# B&R Automation Studio project 2x1HWDemo
Automation Studio 4.9.2.46; technology packages: mapp 5.14.0, mappCockpit 5.14.0, mappControl 5.14.0, mappMotion 5.14.0, mappView 5.14.0

## Configuration 1685

CPU X20CP1685, AutomationRuntime C4.90, Build 6.3.0, Safety 1.10, Vc V4.72.2

### Task classes (Cpu.sw)
```
Cyclic#1 (cycle 1000 us, tolerance 0 us):
  6DCtrl <- Source.6DCtrl.6DCtrl.prg
  RbtCtrl <- Source.Robot.RbtCtrl.prg
  ShCtrl <- Source.ShuttleCtrl.ShCtrl.prg
Cyclic#2 (cycle 10000 us, tolerance 10000 us):
  Main <- Source.Main.Main.prg
Cyclic#4:
  Recovery <- Source.ShuttleCtrl.Recovery.prg
Cyclic#8 (cycle 1000 us):
  Vis <- Source.Auxil.Vis.prg
  AuditCtrl <- Source.Auxil.AuditCtrl.prg
  MacroLoad <- Source.6DCtrl.MacroLoad.prg
DataObjects: McAcpSys
Binaries: mvLoader, arcoal, McMechSys, arflatprv, arsvcreg, McProfGen, TCData, McAcpSim, mCoWebSc, FWRules, McAcpDrv, udbdef, Role, Config_3, arconfig, Settings, User, asfw, ashwd, Config_1, ashwac, sysconf, Config_4, Config, Hierarchy, Config_2, iomap
Libraries: McBase, McAxis, MpBase, AsMath, AsXml, operator, runtime, astime, AsIecCon, standard, AsBrStr, AsIODiag, LoggingLib, asstring, ArEventLog, AsTCP, FileIO, snprintf, brsystem, AsZip, MTTypes, sys_lib, CoTrace, McAcpAx, McPathGen, McAcpTrak, McAxGroup, McProgInt, MpRobotics, MTBasics, McAcp6D, MpAudit, asarlog, asepl, asmem, aruser, dataobj, powerlnk, asarprof, arssl
```

### Hardware
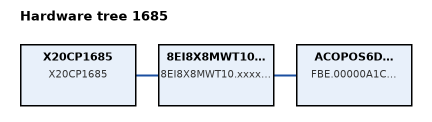
```
8EI8X8MWT10.xxxx-1 : 8EI8X8MWT10.xxxx-1 v2.3.0.2  [PLK1 -> X20CP1685.IF3 (NodeNumber=2) [Cable Type=PowerlinkCable, Length=10, Version=1.0.0.3]; PLK2 -> ACOPOS6D_POWERLINK.PLK1 (NodeNumber=2) [Cable Type=PowerlinkCable, Length=10, Version=1.0.0.3]]
  DriveConfiguration/Module:
    McAcoposTypeID = AcoposP3TConfig
    ActivateACOPOSSimulationOnPLC = 1
  DriveConfiguration/Channel[1]/RealAxis:
    AxisReference = gAxisQ1
  DriveConfiguration/Channel[1]/RealAxis/MechanicalElements/Gearbox:
    InputIsReadOnly = 0
    Input = 1
    OutputIsReadOnly = 0
    Output = 1
  DriveConfiguration/Channel[1]/RealAxis/MechanicalElements/RotaryToLinearTransformation:
    ReferenceDistanceIsReadOnly = 0
    ReferenceDistance = 1
  DriveConfiguration/Channel[1]/RealAxis/Controller:
    ModeIsReadOnly = 0
    Mode = PositionController
  DriveConfiguration/Channel[1]/RealAxis/Controller/Mode/Position:
    ProportionalGain = 50.0
    IntegrationTime = 0.0
    PredictionTime = 0.0004
    TotalDelayTime = 0.0004
  DriveConfiguration/Channel[1]/RealAxis/Controller/Mode/Speed:
    ProportionalGainIsReadOnly = 0
    ProportionalGain = 2.0
    IntegrationTimeIsReadOnly = 0
    IntegrationTime = 0.0
    FilterTimeIsReadOnly = 0
    FilterTime = 0.0
  DriveConfiguration/Channel[1]/RealAxis/Controller/Mode/LoopFilters:
    LoopFilter1 = NotUsed
    LoopFilter2 = NotUsed
    LoopFilter3 = NotUsed
  DriveConfiguration/Channel[1]/RealAxis/Homing:
    Mode = Direct
  DriveConfiguration/Channel[1]/RealAxis/Homing/Mode:
    Position = 0.0
    ReferencePulse = NotUsed
  DriveConfiguration/Channel[1]/RealAxis/Homing:
    RestorePositionVariable = 
  DriveConfiguration/Channel[1]/RealAxis/StopReaction:
    Quickstop = DecelerationLimit
    DriveError = DecelerationLimit
  DriveConfiguration/Channel[1]/RealAxis/MovementErrorLimits:
    PositionError = 1.0
    VelocityErrorMonitoring = Automatic1
  DriveConfiguration/Channel[1]/RealAxis:
    JerkFilter = NotUsed
  DriveConfiguration/Channel[1]/RealAxis/DigitalInputs/HomingSwitch:
    Source = NotUsed
    Level = High
  DriveConfiguration/Channel[1]/RealAxis/DigitalInputs/PositiveLimitSwitch:
    Source = NotUsed
    Level = High
  DriveConfiguration/Channel[1]/RealAxis/DigitalInputs/NegativeLimitSwitch:
    Source = NotUsed
    Level = High
  DriveConfiguration/Channel[1]/RealAxis/DigitalInputs/Trigger1:
    Source = X8Trigger1
    Level = High
  DriveConfiguration/Channel[1]/RealAxis/DigitalInputs/Trigger2:
    Source = X8Trigger2
    Level = High
  DriveConfiguration/Channel[1]/RealAxis/DigitalInputs/Quickstop:
    Input = Trigger2
  DriveConfiguration/Channel[1]/RealAxis/Simulation:
    SimulationModeOnPLC = SetValueGeneration
    SimulationModeOnACOPOS = NotUsed
  DriveConfiguration/Channel[2]/RealAxis:
    AxisReference = gAxisQ2
  DriveConfiguration/Channel[2]/RealAxis/MechanicalElements/Gearbox:
    InputIsReadOnly = 0
    Input = 1
    OutputIsReadOnly = 0
    Output = 1
  DriveConfiguration/Channel[2]/RealAxis/MechanicalElements/RotaryToLinearTransformation:
    ReferenceDistanceIsReadOnly = 0
    ReferenceDistance = 1
  DriveConfiguration/Channel[2]/RealAxis/Controller:
    ModeIsReadOnly = 0
    Mode = PositionController
  DriveConfiguration/Channel[2]/RealAxis/Controller/Mode/Position:
    ProportionalGain = 50.0
    IntegrationTime = 0.0
    PredictionTime = 0.0004
    TotalDelayTime = 0.0004
  DriveConfiguration/Channel[2]/RealAxis/Controller/Mode/Speed:
    ProportionalGainIsReadOnly = 0
    ProportionalGain = 2.0
    IntegrationTimeIsReadOnly = 0
    IntegrationTime = 0.0
    FilterTimeIsReadOnly = 0
    FilterTime = 0.0
  DriveConfiguration/Channel[2]/RealAxis/Controller/Mode/LoopFilters:
    LoopFilter1 = NotUsed
    LoopFilter2 = NotUsed
    LoopFilter3 = NotUsed
  DriveConfiguration/Channel[2]/RealAxis/Homing:
    Mode = Direct
  DriveConfiguration/Channel[2]/RealAxis/Homing/Mode:
    Position = 0.0
    ReferencePulse = NotUsed
  DriveConfiguration/Channel[2]/RealAxis/Homing:
    RestorePositionVariable = 
  DriveConfiguration/Channel[2]/RealAxis/StopReaction:
    Quickstop = DecelerationLimit
    DriveError = DecelerationLimit
  DriveConfiguration/Channel[2]/RealAxis/MovementErrorLimits:
    PositionError = 1.0
    VelocityErrorMonitoring = Automatic1
  DriveConfiguration/Channel[2]/RealAxis:
    JerkFilter = NotUsed
  DriveConfiguration/Channel[2]/RealAxis/DigitalInputs/HomingSwitch:
    Source = NotUsed
    Level = High
  DriveConfiguration/Channel[2]/RealAxis/DigitalInputs/PositiveLimitSwitch:
    Source = NotUsed
    Level = High
  DriveConfiguration/Channel[2]/RealAxis/DigitalInputs/NegativeLimitSwitch:
    Source = NotUsed
    Level = High
  DriveConfiguration/Channel[2]/RealAxis/DigitalInputs/Trigger1:
    Source = X8Trigger1
    Level = High
  DriveConfiguration/Channel[2]/RealAxis/DigitalInputs/Trigger2:
    Source = X8Trigger2
    Level = High
  DriveConfiguration/Channel[2]/RealAxis/DigitalInputs/Quickstop:
    Input = Trigger2
  DriveConfiguration/Channel[2]/RealAxis/Simulation:
    SimulationModeOnPLC = SetValueGeneration
    SimulationModeOnACOPOS = NotUsed
  DriveConfiguration/Channel[3]/RealAxis:
    AxisReference = gAxisQ3
  DriveConfiguration/Channel[3]/RealAxis/MechanicalElements/Gearbox:
    InputIsReadOnly = 0
    Input = 1
    OutputIsReadOnly = 0
    Output = 1
  DriveConfiguration/Channel[3]/RealAxis/MechanicalElements/RotaryToLinearTransformation:
    ReferenceDistanceIsReadOnly = 0
    ReferenceDistance = 1
  DriveConfiguration/Channel[3]/RealAxis/Controller:
    ModeIsReadOnly = 0
    Mode = PositionController
  DriveConfiguration/Channel[3]/RealAxis/Controller/Mode/Position:
    ProportionalGain = 50.0
    IntegrationTime = 0.0
    PredictionTime = 0.0004
    TotalDelayTime = 0.0004
  DriveConfiguration/Channel[3]/RealAxis/Controller/Mode/Speed:
    ProportionalGainIsReadOnly = 0
    ProportionalGain = 2.0
    IntegrationTimeIsReadOnly = 0
    IntegrationTime = 0.0
    FilterTimeIsReadOnly = 0
    FilterTime = 0.0
  DriveConfiguration/Channel[3]/RealAxis/Controller/Mode/LoopFilters:
    LoopFilter1 = NotUsed
    LoopFilter2 = NotUsed
    LoopFilter3 = NotUsed
  DriveConfiguration/Channel[3]/RealAxis/Homing:
    Mode = Direct
  DriveConfiguration/Channel[3]/RealAxis/Homing/Mode:
    Position = 0.0
    ReferencePulse = NotUsed
  DriveConfiguration/Channel[3]/RealAxis/Homing:
    RestorePositionVariable = 
  DriveConfiguration/Channel[3]/RealAxis/StopReaction:
    Quickstop = DecelerationLimit
    DriveError = DecelerationLimit
  DriveConfiguration/Channel[3]/RealAxis/MovementErrorLimits:
    PositionError = 1.0
    VelocityErrorMonitoring = Automatic1
  DriveConfiguration/Channel[3]/RealAxis:
    JerkFilter = NotUsed
  DriveConfiguration/Channel[3]/RealAxis/DigitalInputs/HomingSwitch:
    Source = NotUsed
    Level = High
  DriveConfiguration/Channel[3]/RealAxis/DigitalInputs/PositiveLimitSwitch:
    Source = NotUsed
    Level = High
  DriveConfiguration/Channel[3]/RealAxis/DigitalInputs/NegativeLimitSwitch:
    Source = NotUsed
    Level = High
  DriveConfiguration/Channel[3]/RealAxis/DigitalInputs/Trigger1:
    Source = X8Trigger1
    Level = High
  DriveConfiguration/Channel[3]/RealAxis/DigitalInputs/Trigger2:
    Source = X8Trigger2
    Level = High
  DriveConfiguration/Channel[3]/RealAxis/DigitalInputs/Quickstop:
    Input = Trigger2
  DriveConfiguration/Channel[3]/RealAxis/Simulation:
    SimulationModeOnPLC = SetValueGeneration
    SimulationModeOnACOPOS = NotUsed
ACOPOS6D_POWERLINK : FBE.00000A1C_PlanarMotorIncorporatedPOWERLINK v1.12.05 (OrderNumber=Planar Motor Incorporated POWERLINK)  [PLK1 -> 8EI8X8MWT10.xxxx-1.PLK2 (NodeNumber=1) [Cable Type=PowerlinkCable, Length=10, Version=1.0.0.3]]
  Supervision = off
X20CP1685 : X20CP1685 v1.1.0.0
  Connector IF2:
    ActivateDevice = 1
  Connector IF3:
    CycleTime = 1000
  ConfigurationID = OnsiteDemo_1685
  UserPartitionSize = 10
  TimerDeviceType = EPLX2X
  TimerDevice = X20CP1685.IF3
  Cyclic1Duration = 1000
  Cyclic1Tolerance = 0
  Cyclic2Duration = 10000
  Cyclic2Tolerance = 10000
  Cyclic8Duration = 1000
  FtpUser1
  FtpUsername1 = user
  FtpUserPassword1 = OnC+KhD/SpTljM37peNi/Txa+vmo0PgBkRCvsZXBTJk=  // user
  FtpUserSalt1 = 0mgKB/Te
  FTPAccessRight1 = 0
  ActivateOpcUa = 1
  OpcUaInformationModels_PV_Version = 2
```

## Configuration 2200

CPU 5APC2100.BY48-000, AutomationRuntime B4.82, Build 6.3.0, Safety 1.10, Vc V4.72.2

### Task classes (Cpu.sw)
```
Cyclic#1 (cycle 1000 us, tolerance 0 us):
  6DCtrl <- Source.6DCtrl.6DCtrl.prg
  ShCtrl <- Source.ShuttleCtrl.ShCtrl.prg
  RbtCtrl <- Source.Robot.RbtCtrl.prg
Cyclic#2 (cycle 10000 us, tolerance 10000 us):
  Main <- Source.Main.Main.prg
Cyclic#4:
  Recovery <- Source.ShuttleCtrl.Recovery.prg
Cyclic#8 (cycle 2000 us):
  Vis <- Source.Auxil.Vis.prg
  AuditCtrl <- Source.Auxil.AuditCtrl.prg
  MacroLoad <- Source.6DCtrl.MacroLoad.prg
DataObjects: McAcpSys
Binaries: mvLoader, arcoal, McMechSys, arflatprv, arsvcreg, McProfGen, TCData, McAcpSim, mCoWebSc, FWRules, McAcpDrv, udbdef, Role, Config_3, arconfig, Settings, User, asfw, ashwd, Config_1, ashwac, sysconf, Config_4, Config, Hierarchy, Config_2, iomap
Libraries: McBase, McAxis, MpBase, AsMath, AsXml, operator, runtime, astime, AsIecCon, standard, AsBrStr, AsIODiag, LoggingLib, asstring, ArEventLog, AsTCP, FileIO, snprintf, brsystem, AsZip, MTTypes, sys_lib, CoTrace, McAcpAx, McPathGen, McAcpTrak, McAxGroup, McProgInt, MpRobotics, MTBasics, McAcp6D, MpAudit, asarlog, asepl, asmem, aruser, dataobj, powerlnk, asarprof, arssl, MTFilter
```

### Hardware
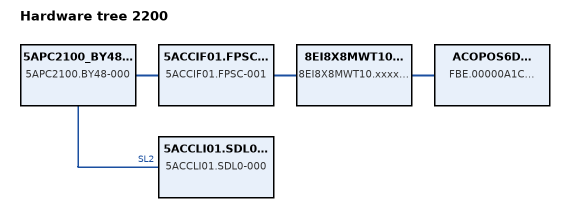
```
5ACCIF01.FPSC-001 : 5ACCIF01.FPSC-001 v1.8.1.0  [SL -> 5APC2100_BY48_000.SL1]
  Connector IF1:
    CycleTime = 1000
5ACCLI01.SDL0-000 : 5ACCLI01.SDL0-000 v2.0.0.0  [SL -> 5APC2100_BY48_000.SL2]
5APC2100_BY48_000 : 5APC2100.BY48-000 v2.1.0.0
  Connector IF3:
    AssignedOperatingSystem = ARemb
    ActivateDevice = 1
    Mode = Manual
    InternetAddress = 192.168.10.85
    SubnetMask = 255.255.255.0
    ActivateSnmp = 2
  Connector IF4:
    AssignedOperatingSystem = ARemb
    ActivateDevice = 1
    Mode = Manual
    InternetAddress = 192.168.1.69
    SubnetMask = 255.255.255.0
  Connector IF5:
    AssignedOperatingSystem = ARemb
  Connector IF6:
    AssignedOperatingSystem = ARemb
  ConfigurationID = OnsiteDemo_1685
  UserPartitionSize = 10
  AutomaticTransferOfUserfiles = on
  TimerDeviceType = EPLX2X
  TimerDevice = 5ACCIF01.FPSC-001.IF1
  Cyclic1Duration = 1000
  Cyclic1Tolerance = 0
  Cyclic2Duration = 10000
  Cyclic2Tolerance = 10000
  Cyclic8Duration = 2000
  FileDevice1
  FileDeviceName1 = CNC_PrgDir
  FileDevicePath1 = F:/Programs
  FileDevice2
  FileDeviceName2 = 6DMacro
  FileDevicePath2 = F:/Macros
  FtpUser1
  FtpUsername1 = user
  FtpUserPassword1 = OnC+KhD/SpTljM37peNi/Txa+vmo0PgBkRCvsZXBTJk=  // user
  FtpUserSalt1 = 0mgKB/Te
  FTPAccessRight1 = 0
  ActivateOpcUa = 1
  OpcUaInformationModels_PV_Version = 2
8EI8X8MWT10.xxxx-1 : 8EI8X8MWT10.xxxx-1 v2.3.0.2  [PLK1 -> 5ACCIF01.FPSC-001.IF1 (NodeNumber=2) [Cable Type=PowerlinkCable, Length=10, Version=1.0.0.3]; PLK2 -> ACOPOS6D_POWERLINK.PLK1 (NodeNumber=2) [Cable Type=PowerlinkCable, Length=10, Version=1.0.0.3]]
  DriveConfiguration/Module:
    McAcoposTypeID = AcoposP3TConfig
    ActivateACOPOSSimulationOnPLC = 1
  DriveConfiguration/Channel[1]/RealAxis:
    AxisReference = gAxisQ1
  DriveConfiguration/Channel[1]/RealAxis/MechanicalElements/Gearbox:
    InputIsReadOnly = 0
    Input = 1
    OutputIsReadOnly = 0
    Output = 1
  DriveConfiguration/Channel[1]/RealAxis/MechanicalElements/RotaryToLinearTransformation:
    ReferenceDistanceIsReadOnly = 0
    ReferenceDistance = 1
  DriveConfiguration/Channel[1]/RealAxis/Controller:
    ModeIsReadOnly = 0
    Mode = PositionController
  DriveConfiguration/Channel[1]/RealAxis/Controller/Mode/Position:
    ProportionalGain = 50.0
    IntegrationTime = 0.0
    PredictionTime = 0.0004
    TotalDelayTime = 0.0004
  DriveConfiguration/Channel[1]/RealAxis/Controller/Mode/Speed:
    ProportionalGainIsReadOnly = 0
    ProportionalGain = 2.0
    IntegrationTimeIsReadOnly = 0
    IntegrationTime = 0.0
    FilterTimeIsReadOnly = 0
    FilterTime = 0.0
  DriveConfiguration/Channel[1]/RealAxis/Controller/Mode/LoopFilters:
    LoopFilter1 = NotUsed
    LoopFilter2 = NotUsed
    LoopFilter3 = NotUsed
  DriveConfiguration/Channel[1]/RealAxis/Homing:
    Mode = Direct
  DriveConfiguration/Channel[1]/RealAxis/Homing/Mode:
    Position = 0.0
    ReferencePulse = NotUsed
  DriveConfiguration/Channel[1]/RealAxis/Homing:
    RestorePositionVariable = 
  DriveConfiguration/Channel[1]/RealAxis/StopReaction:
    Quickstop = DecelerationLimit
    DriveError = DecelerationLimit
  DriveConfiguration/Channel[1]/RealAxis/MovementErrorLimits:
    PositionError = 1.0
    VelocityErrorMonitoring = Automatic1
  DriveConfiguration/Channel[1]/RealAxis:
    JerkFilter = NotUsed
  DriveConfiguration/Channel[1]/RealAxis/DigitalInputs/HomingSwitch:
    Source = NotUsed
    Level = High
  DriveConfiguration/Channel[1]/RealAxis/DigitalInputs/PositiveLimitSwitch:
    Source = NotUsed
    Level = High
  DriveConfiguration/Channel[1]/RealAxis/DigitalInputs/NegativeLimitSwitch:
    Source = NotUsed
    Level = High
  DriveConfiguration/Channel[1]/RealAxis/DigitalInputs/Trigger1:
    Source = X8Trigger1
    Level = High
  DriveConfiguration/Channel[1]/RealAxis/DigitalInputs/Trigger2:
    Source = X8Trigger2
    Level = High
  DriveConfiguration/Channel[1]/RealAxis/DigitalInputs/Quickstop:
    Input = Trigger2
  DriveConfiguration/Channel[1]/RealAxis/Simulation:
    SimulationModeOnPLC = SetValueGeneration
    SimulationModeOnACOPOS = NotUsed
  DriveConfiguration/Channel[2]/RealAxis:
    AxisReference = gAxisQ2
  DriveConfiguration/Channel[2]/RealAxis/MechanicalElements/Gearbox:
    InputIsReadOnly = 0
    Input = 1
    OutputIsReadOnly = 0
    Output = 1
  DriveConfiguration/Channel[2]/RealAxis/MechanicalElements/RotaryToLinearTransformation:
    ReferenceDistanceIsReadOnly = 0
    ReferenceDistance = 1
  DriveConfiguration/Channel[2]/RealAxis/Controller:
    ModeIsReadOnly = 0
    Mode = PositionController
  DriveConfiguration/Channel[2]/RealAxis/Controller/Mode/Position:
    ProportionalGain = 50.0
    IntegrationTime = 0.0
    PredictionTime = 0.0004
    TotalDelayTime = 0.0004
  DriveConfiguration/Channel[2]/RealAxis/Controller/Mode/Speed:
    ProportionalGainIsReadOnly = 0
    ProportionalGain = 2.0
    IntegrationTimeIsReadOnly = 0
    IntegrationTime = 0.0
    FilterTimeIsReadOnly = 0
    FilterTime = 0.0
  DriveConfiguration/Channel[2]/RealAxis/Controller/Mode/LoopFilters:
    LoopFilter1 = NotUsed
    LoopFilter2 = NotUsed
    LoopFilter3 = NotUsed
  DriveConfiguration/Channel[2]/RealAxis/Homing:
    Mode = Direct
  DriveConfiguration/Channel[2]/RealAxis/Homing/Mode:
    Position = 0.0
    ReferencePulse = NotUsed
  DriveConfiguration/Channel[2]/RealAxis/Homing:
    RestorePositionVariable = 
  DriveConfiguration/Channel[2]/RealAxis/StopReaction:
    Quickstop = DecelerationLimit
    DriveError = DecelerationLimit
  DriveConfiguration/Channel[2]/RealAxis/MovementErrorLimits:
    PositionError = 1.0
    VelocityErrorMonitoring = Automatic1
  DriveConfiguration/Channel[2]/RealAxis:
    JerkFilter = NotUsed
  DriveConfiguration/Channel[2]/RealAxis/DigitalInputs/HomingSwitch:
    Source = NotUsed
    Level = High
  DriveConfiguration/Channel[2]/RealAxis/DigitalInputs/PositiveLimitSwitch:
    Source = NotUsed
    Level = High
  DriveConfiguration/Channel[2]/RealAxis/DigitalInputs/NegativeLimitSwitch:
    Source = NotUsed
    Level = High
  DriveConfiguration/Channel[2]/RealAxis/DigitalInputs/Trigger1:
    Source = X8Trigger1
    Level = High
  DriveConfiguration/Channel[2]/RealAxis/DigitalInputs/Trigger2:
    Source = X8Trigger2
    Level = High
  DriveConfiguration/Channel[2]/RealAxis/DigitalInputs/Quickstop:
    Input = Trigger2
  DriveConfiguration/Channel[2]/RealAxis/Simulation:
    SimulationModeOnPLC = SetValueGeneration
    SimulationModeOnACOPOS = NotUsed
  DriveConfiguration/Channel[3]/RealAxis:
    AxisReference = gAxisQ3
  DriveConfiguration/Channel[3]/RealAxis/MechanicalElements/Gearbox:
    InputIsReadOnly = 0
    Input = 1
    OutputIsReadOnly = 0
    Output = 1
  DriveConfiguration/Channel[3]/RealAxis/MechanicalElements/RotaryToLinearTransformation:
    ReferenceDistanceIsReadOnly = 0
    ReferenceDistance = 1
  DriveConfiguration/Channel[3]/RealAxis/Controller:
    ModeIsReadOnly = 0
    Mode = PositionController
  DriveConfiguration/Channel[3]/RealAxis/Controller/Mode/Position:
    ProportionalGain = 50.0
    IntegrationTime = 0.0
    PredictionTime = 0.0004
    TotalDelayTime = 0.0004
  DriveConfiguration/Channel[3]/RealAxis/Controller/Mode/Speed:
    ProportionalGainIsReadOnly = 0
    ProportionalGain = 2.0
    IntegrationTimeIsReadOnly = 0
    IntegrationTime = 0.0
    FilterTimeIsReadOnly = 0
    FilterTime = 0.0
  DriveConfiguration/Channel[3]/RealAxis/Controller/Mode/LoopFilters:
    LoopFilter1 = NotUsed
    LoopFilter2 = NotUsed
    LoopFilter3 = NotUsed
  DriveConfiguration/Channel[3]/RealAxis/Homing:
    Mode = Direct
  DriveConfiguration/Channel[3]/RealAxis/Homing/Mode:
    Position = 0.0
    ReferencePulse = NotUsed
  DriveConfiguration/Channel[3]/RealAxis/Homing:
    RestorePositionVariable = 
  DriveConfiguration/Channel[3]/RealAxis/StopReaction:
    Quickstop = DecelerationLimit
    DriveError = DecelerationLimit
  DriveConfiguration/Channel[3]/RealAxis/MovementErrorLimits:
    PositionError = 1.0
    VelocityErrorMonitoring = Automatic1
  DriveConfiguration/Channel[3]/RealAxis:
    JerkFilter = NotUsed
  DriveConfiguration/Channel[3]/RealAxis/DigitalInputs/HomingSwitch:
    Source = NotUsed
    Level = High
  DriveConfiguration/Channel[3]/RealAxis/DigitalInputs/PositiveLimitSwitch:
    Source = NotUsed
    Level = High
  DriveConfiguration/Channel[3]/RealAxis/DigitalInputs/NegativeLimitSwitch:
    Source = NotUsed
    Level = High
  DriveConfiguration/Channel[3]/RealAxis/DigitalInputs/Trigger1:
    Source = X8Trigger1
    Level = High
  DriveConfiguration/Channel[3]/RealAxis/DigitalInputs/Trigger2:
    Source = X8Trigger2
    Level = High
  DriveConfiguration/Channel[3]/RealAxis/DigitalInputs/Quickstop:
    Input = Trigger2
  DriveConfiguration/Channel[3]/RealAxis/Simulation:
    SimulationModeOnPLC = SetValueGeneration
    SimulationModeOnACOPOS = NotUsed
ACOPOS6D_POWERLINK : FBE.00000A1C_PlanarMotorIncorporatedPOWERLINK v1.12.05 (OrderNumber=Planar Motor Incorporated POWERLINK)  [PLK1 -> 8EI8X8MWT10.xxxx-1.PLK2 (NodeNumber=1) [Cable Type=PowerlinkCable, Length=10, Version=1.0.0.3]]
  Supervision = off
```

### Config_2.axis - 5APC2100_BY48_000/mappMotion/Robot/3AxesDeltaA/Config_2.axis
```
Element gAxisQ1 (Type=axis)
  BaseTypeIsReadOnly = 0
  BaseType = RotaryBounded
    MeasurementUnitIsReadOnly = 0
    MeasurementUnit = 17476
    MeasurementResolutionIsReadOnly = 0
    MeasurementResolution = 0.01
    CountDirectionIsReadOnly = 0
    CountDirection = Standard
  MovementLimitsIsReadOnly = 0
  MovementLimits = Internal
    Position:
      LowerLimitMin = -1.79769313486231E308
      UpperLimitMax = 1.79769313486231E308
      LowerLimit = -1000.0
      UpperLimit = 1000.0
    VelocityIsReadOnly = 0
    Velocity:
      VelocityMax = 3.4E38
      Velocity = 100.0
    AccelerationIsReadOnly = 0
    Acceleration:
      AccelerationMax = 3.4E38
      Acceleration = 500.0
    DecelerationIsReadOnly = 0
    Deceleration:
      DecelerationMax = 3.4E38
      Deceleration = 500.0
  Alarms = None
Element gAxisQ2 (Type=axis)
  BaseTypeIsReadOnly = 0
  BaseType = RotaryBounded
    MeasurementUnitIsReadOnly = 0
    MeasurementUnit = 17476
    MeasurementResolutionIsReadOnly = 0
    MeasurementResolution = 0.01
    CountDirectionIsReadOnly = 0
    CountDirection = Standard
  MovementLimitsIsReadOnly = 0
  MovementLimits = Internal
    Position:
      LowerLimitMin = -1.79769313486231E308
      UpperLimitMax = 1.79769313486231E308
      LowerLimit = -1000.0
      UpperLimit = 1000.0
    VelocityIsReadOnly = 0
    Velocity:
      VelocityMax = 3.4E38
      Velocity = 100.0
    AccelerationIsReadOnly = 0
    Acceleration:
      AccelerationMax = 3.4E38
      Acceleration = 500.0
    DecelerationIsReadOnly = 0
    Deceleration:
      DecelerationMax = 3.4E38
      Deceleration = 500.0
  Alarms = None
Element gAxisQ3 (Type=axis)
  BaseTypeIsReadOnly = 0
  BaseType = RotaryBounded
    MeasurementUnitIsReadOnly = 0
    MeasurementUnit = 17476
    MeasurementResolutionIsReadOnly = 0
    MeasurementResolution = 0.01
    CountDirectionIsReadOnly = 0
    CountDirection = Standard
  MovementLimitsIsReadOnly = 0
  MovementLimits = Internal
    Position:
      LowerLimitMin = -1.79769313486231E308
      UpperLimitMax = 1.79769313486231E308
      LowerLimit = -1000.0
      UpperLimit = 1000.0
    VelocityIsReadOnly = 0
    Velocity:
      VelocityMax = 3.4E38
      Velocity = 100.0
    AccelerationIsReadOnly = 0
    Acceleration:
      AccelerationMax = 3.4E38
      Acceleration = 500.0
    DecelerationIsReadOnly = 0
    Deceleration:
      DecelerationMax = 3.4E38
      Deceleration = 500.0
  Alarms = None
```

### Config_3.mechanicalsystem - 5APC2100_BY48_000/mappMotion/Robot/3AxesDeltaA/Config_3.mechanicalsystem
```
Element MechSys_3AxDeltaA (Type=mechanicalsystem)
  Type = Delta
    Subtype = 3AxesDeltaA
      Description = Standard
        Dimensions:
          BasePlatform:
            CenterIsReadOnly = 0
            Center:
              X = 0.0
              Y = 0.0
              Z = -267.0
            ArmLinkPointIsReadOnly = 0
            Arm1LinkPoint:
              Angle = 0.0
              Radius = 205
              Z = 0.0
            Arm2LinkPoint:
              Angle = 120.0
              Radius = 205
              Z = 0.0
            Arm3LinkPoint:
              Angle = 240.0
              Radius = 205.0
              Z = 0.0
          Arms:
            ArmIsReadOnly = 0
            Arm1:
              UpperArmLength = 430.0
              LowerArmLength = 1105.0
            Arm2:
              UpperArmLength = 430.0
              LowerArmLength = 1105.0
            Arm3:
              UpperArmLength = 430.0
              LowerArmLength = 1105.0
          EndEffectorPlatform:
            ArmLinkPointIsReadOnly = 0
            Arm1LinkPoint:
              Radius = 50.0
              Z = 0.0
            Arm2LinkPoint:
              Radius = 50.0
              Z = 0.0
            Arm3LinkPoint:
              Radius = 50.0
              Z = 0.0
            TranslationToFlange:
              X = 0.0
              Y = 0.0
              Z = -50
        Offsets:
          JointAxisIsReadOnly = 0
          JointAxis[1] = 0.0
          JointAxis[2] = 0.0
          JointAxis[3] = 0.0
        CountDirections:
          JointAxisIsReadOnly = 0
          JointAxis[1] = Standard
          JointAxis[2] = Standard
          JointAxis[3] = Standard
      CoordinatesNames = Default
        XCoordinateName = X
        YCoordinateName = Y
        ZCoordinateName = Z
      WireFrameModel = Standard
        UpperArm1 = ConnectionLine
          Distance = 0.0
        LowerArm1 = ConnectionLine
          Distance = 0.0
        UpperArm2 = ConnectionLine
          Distance = 0.0
        LowerArm2 = ConnectionLine
          Distance = 0.0
        UpperArm3 = ConnectionLine
          Distance = 0.0
        LowerArm3 = ConnectionLine
          Distance = 0.0
        EndEffectorPlatformToFlange = ConnectionLine
          Distance = 0.0
        FlangeToTcp = ConnectionLine
          Distance = 0.0
      DynamicModel = DynParTable
        TableRef
      InternalDynamicModel = NotUsed
      JointAxesPositionLimits:
        JointAxis[1] = UseAxisLimits
        JointAxis[2] = UseAxisLimits
        JointAxis[3] = UseAxisLimits
```

### Config_4.axesgroupfeature - 5APC2100_BY48_000/mappMotion/Robot/3AxesDeltaA/Config_4.axesgroupfeature
```
Element Feature_Programs (Type=axesgroupfeature)
  Type = Program
    ModalDataBehaviour = UseAxesGroupSettings
    InitialSettings:
      InterpolationTypes = LinearRapid
      PositionCoordinates = Absolute
      CircleCoordinates = Relative
      JACS_ACSProgramming = JACS
      ContourConnection = Inactive
      ProgrammingUnits = UseAxesGroupSettings
      Feedrates:
        FeedPath = Standard
        FeedCharacteristic = StandardCharacteristic
        FeedType = Feedrate
        FeedReduction = Inactive
        FeedrateValue = 0.0
        InverseFeedrateValue = 0.0
        FeedratePerRevValue = 0.0
    DefaultLanguage = BRGCode
    Location = Default
      FileDevice = CNC_PrgDir
Element Feature_Jogging (Type=axesgroupfeature)
  Type = Jogging
Element Feature_Frames (Type=axesgroupfeature)
  Type = FrameHierarchy
    ModalDataBehaviour = UseAxesGroupSettings
    FrameHierarchy = Custom
      FramePropertyMapping:
        BCS = RobotBase
        PCS = RobotBase
        SCS1 = 
        SCS2
        SCS3
        SCS4
        SCS5
      MCS:
        Frame[1]:
          Name = RobotBase
          Type = StandardFrame
            Translation:
              X = 240.0
              Y = 0.0
              Z = 1425.0
            Orientation:
              Angle1 = 0.0
              Angle2 = 0.0
              Angle3 = 0.0
        Frame[2]:
          Name = TrakSync
          Type = StandardFrame
            Translation:
              X = 120
              Y = 0.0
              Z = 90
            Orientation:
              Angle1 = 0.0
              Angle2 = 0.0
              Angle3 = 0
```

## Configuration 910

CPU 5PC900.TS17-00, AutomationRuntime C4.90, Build 6.3.0, Safety 0.0, Vc V4.72.2

### Task classes (Cpu.sw)
```
Cyclic#1 (cycle 1000 us, tolerance 0 us):
  6DCtrl <- Source.6DCtrl.6DCtrl.prg
  ShCtrl <- Source.ShuttleCtrl.ShCtrl.prg
  KalmanTes1 <- (binary)
Cyclic#2 (cycle 5000 us):
  MacroDemo <- Source.Demos.MacroDemo.prg
  VariedMovD <- Source.Demos.VariedMovDemo.prg
  KalmanTest <- Source.ShuttleCtrl.KalmanTesting.prg
Cyclic#3:
  Main <- Source.Main.Main.prg
Cyclic#4:
  Recovery <- Source.ShuttleCtrl.Recovery.prg
  GenMoveDem <- Source.Demos.GenMoveDemo.prg
Cyclic#8 (cycle 2000 us):
  AuditCtrl <- Source.Auxil.AuditCtrl.prg
  MacroLoad <- Source.6DCtrl.MacroLoad.prg
  Vis <- Source.Auxil.Vis.prg
Binaries: TCLang, udbdef, FWRules, mvLoader, mCoWebSc, TCData, OpcUaSrv, arsvcreg, mcacpdrv, arflatprv, arcoal, iomap, asfw, Role, ashwd, sysconf, arconfig, ashwac, User, Config, TC, Config_1, TraceConfi, Settings
Libraries: MpAudit, MpBase, MpRobotics, McAxGroup, McBase, McPathGen, McAcpAx, McAcpTrak, McAxis, McProgInt, CoTrace, AsZip, FileIO, runtime, MTBasics, brsystem, MTFilter, sys_lib, MTTypes, operator, astime, AsIecCon, standard, McAcp6D, AsXml, AsBrStr, AsIODiag, LoggingLib, asstring, ArEventLog, AsTCP, snprintf, MpFile, MpServer, WFilter, AsBrMath, asmem, arssl, asio, asarprof, powerlnk, dataobj, aruser, asepl, asarlog, asusb, asmath
```

### Hardware
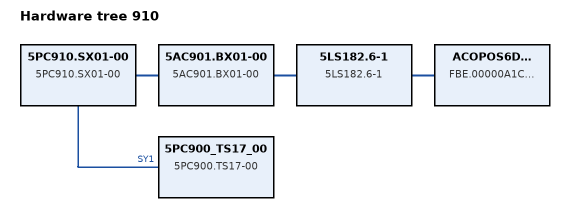
```
5AC901.BX01-00 : 5AC901.BX01-00 v1.0.1.0  [SY -> 5PC910.SX01-00.SY3]
5LS182.6-1 : 5LS182.6-1 v1.3.1.0  [SL -> 5AC901.BX01-00.SL1]
  Connector IF1:
    CycleTime = 1000
5PC900_TS17_00 : 5PC900.TS17-00 v2.1.0.0  [SY -> 5PC910.SX01-00.SY1]
  ConfigurationID = OnsiteDemo_910
  UserPartitionSize = 10
  UserRamDevice = PCI.1.LS182.SRAM
  UserRamSize = 500000
  TimerDeviceType = EPLX2X
  TimerDevice = 5LS182.6-1.IF1
  Cyclic1Duration = 1000
  Cyclic1Tolerance = 0
  Cyclic2Duration = 5000
  Cyclic8Duration = 2000
  FileDevice1
  FileDeviceName1 = 6DMacro
  FileDevicePath1 = F:\Macros
  FtpUser1
  FtpUsername1 = user  // user
  FtpUserPassword1 = uWQ3MCiALScWh+25zsAuoOpgOm0XOB8wRCPxpHYIgE4=  // user
  FtpUserSalt1 = pXahafUb
  FTPAccessRight1 = 0
  FTPdevice1 = ALL
  ActivateOpcUa = 1
  OpcUaPort = 4841
  OpcUaInformationModels_PV_Version = 2
5PC910.SX01-00 : 5PC910.SX01-00 v2.1.0.0
  Connector IF1:
    AssignedOperatingSystem = ARemb
  Connector IF3:
    AssignedOperatingSystem = ARemb
    ActivateDevice = 1
    ActivateSnmp = 2
  Connector IF4:
    AssignedOperatingSystem = ARemb
    ActivateDevice = 1
  Connector IF5:
    AssignedOperatingSystem = ARemb
  Connector IF6:
    AssignedOperatingSystem = ARemb
  Connector IF7:
    AssignedOperatingSystem = ARemb
  Connector IF8:
    AssignedOperatingSystem = ARemb
  Connector IF9:
    AssignedOperatingSystem = ARemb
ACOPOS6D_POWERLINK : FBE.00000A1C_PlanarMotorIncorporatedPOWERLINK v1.12.05 (OrderNumber=Planar Motor Incorporated POWERLINK)  [PLK1 -> 5LS182.6-1.IF1 (NodeNumber=1) [Cable Type=PowerlinkCable, Length=10, Version=1.0.0.3]]
  Supervision = off
```

### Config_1.mpfilemanager - 5PC900_TS17_00/mappServices/Config_1.mpfilemanager
```
Element FileManagement (Type=mpfilemanager)
  FileManager:
    Devices:
      0:
        DeviceName = 6DMacro
        Text = Macros
    Access:
      0:
        Folder = *
        Roles:
          0:
            Role = Everyone
            Rights:
              Visible = TRUE
              FolderRead = TRUE
              FileRead = TRUE
              FileEdit = TRUE
              FolderEdit = TRUE
```

## Configuration Config1

CPU 5APC3100.KBU3-000, AutomationRuntime C4.90, Build 6.3.0, Safety 0.0, Vc V4.72.1

### Task classes (Cpu.sw)
```
DataObjects: McAcpSys
Binaries: FWRules, udbdef, McAcpDrv, arsvcreg, McAcpSim, TCData, arflatprv, McMechSys, arcoal, mvLoader, mCoWebSc, arconfig, User, Role, CfgAssbly, sysconf, CfgShuttle, iomap, asfw, ashwac, ashwd, CfgProcPt, CfgSector, Config_3, Settings, Config_1, Config_4, Hierarchy, Config_2
Libraries: McBase, McAcpTrak, McAxis, standard, AsBrStr, AsIODiag, runtime, LoggingLib, astime, asstring, ArEventLog, AsTCP, FileIO, McAxGroup, McPathGen, McProgInt, McAcpAx, snprintf, MpRobotics, MpBase, brsystem, CoTrace, AsZip, MTBasics, MTTypes, sys_lib, powerlnk, asieccon, asarprof, asarlog, asmem, asepl, dataobj, arssl
```

### Hardware
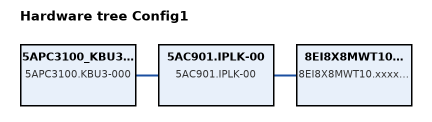
```
5AC901.IPLK-00 : 5AC901.IPLK-00 v1.6.0.0  [SL -> 5APC3100_KBU3_000.SL2]
  Connector IF1:
    DNAConfiguration = manual
    CycleTime = 400
5APC3100_KBU3_000 : 5APC3100.KBU3-000 v2.0.3.0
  Connector IF3:
    AssignedOperatingSystem = ARemb
    ActivateDevice = 1
  Connector IF4:
    AssignedOperatingSystem = ARemb
    ActivateDevice = 1
  Connector IF5:
    AssignedOperatingSystem = ARemb
  Connector IF6:
    AssignedOperatingSystem = ARemb
  Connector IF7:
    AssignedOperatingSystem = ARemb
  Connector IF8:
    AssignedOperatingSystem = ARemb
  ConfigurationID = CustomTracking_Config1
  Simulation = 1
  TimerDeviceType = EPLX2X
  TimerDevice = 5AC901.IPLK-00.IF1
  TaskClassIdleTime = 800
  Cyclic1Duration = 400
  Cyclic1Tolerance = 0
  Cyclic1Output = 1
  Cyclic2Duration = 1600
  Cyclic2Tolerance = 19200
  Cyclic8Duration = 1200
  FileDevice1
  FileDeviceName1 = SvgData
  FileDevicePath1 = ../../../../Logical/Scene/Generated
  FileDevice2
  FileDeviceName2 = CNC_PrgDir
  FileDevicePath2 = ../../../../Logical/Programs
  ActivateOpcUa = 1
  OpcUaInformationModels_PV_Version = 1
8EI8X8MWT10.xxxx-1 : 8EI8X8MWT10.xxxx-1 v2.3.0.2  [PLK2 -> 5AC901.IPLK-00.IF1 (NodeNumber=1) [Cable Type=PowerlinkCable, Length=10, Version=1.0.0.3]]
  DriveConfiguration/Module:
    McAcoposTypeID = AcoposP3TConfig
    ActivateACOPOSSimulationOnPLC = 0
  DriveConfiguration/Channel[1]/RealAxis:
    AxisReference = gAxisQ1
  DriveConfiguration/Channel[1]/RealAxis/MechanicalElements/Gearbox:
    InputIsReadOnly = 0
    Input = 1
    OutputIsReadOnly = 0
    Output = 1
  DriveConfiguration/Channel[1]/RealAxis/MechanicalElements/RotaryToLinearTransformation:
    ReferenceDistanceIsReadOnly = 0
    ReferenceDistance = 1
  DriveConfiguration/Channel[1]/RealAxis/Controller:
    ModeIsReadOnly = 0
    Mode = PositionController
  DriveConfiguration/Channel[1]/RealAxis/Controller/Mode/Position:
    ProportionalGain = 50.0
    IntegrationTime = 0.0
    PredictionTime = 0.0004
    TotalDelayTime = 0.0004
  DriveConfiguration/Channel[1]/RealAxis/Controller/Mode/Speed:
    ProportionalGainIsReadOnly = 0
    ProportionalGain = 2.0
    IntegrationTimeIsReadOnly = 0
    IntegrationTime = 0.0
    FilterTimeIsReadOnly = 0
    FilterTime = 0.0
  DriveConfiguration/Channel[1]/RealAxis/Controller/Mode/LoopFilters:
    LoopFilter1 = NotUsed
    LoopFilter2 = NotUsed
    LoopFilter3 = NotUsed
  DriveConfiguration/Channel[1]/RealAxis/Homing:
    Mode = Direct
  DriveConfiguration/Channel[1]/RealAxis/Homing/Mode:
    Position = 0.0
    ReferencePulse = NotUsed
  DriveConfiguration/Channel[1]/RealAxis/Homing:
    RestorePositionVariable = 
  DriveConfiguration/Channel[1]/RealAxis/StopReaction:
    Quickstop = DecelerationLimit
    DriveError = DecelerationLimit
  DriveConfiguration/Channel[1]/RealAxis/MovementErrorLimits:
    PositionError = 1.0
    VelocityErrorMonitoring = Automatic1
  DriveConfiguration/Channel[1]/RealAxis:
    JerkFilter = NotUsed
  DriveConfiguration/Channel[1]/RealAxis/DigitalInputs/HomingSwitch:
    Source = NotUsed
    Level = High
  DriveConfiguration/Channel[1]/RealAxis/DigitalInputs/PositiveLimitSwitch:
    Source = NotUsed
    Level = High
  DriveConfiguration/Channel[1]/RealAxis/DigitalInputs/NegativeLimitSwitch:
    Source = NotUsed
    Level = High
  DriveConfiguration/Channel[1]/RealAxis/DigitalInputs/Trigger1:
    Source = X8Trigger1
    Level = High
  DriveConfiguration/Channel[1]/RealAxis/DigitalInputs/Trigger2:
    Source = X8Trigger2
    Level = High
  DriveConfiguration/Channel[1]/RealAxis/DigitalInputs/Quickstop:
    Input = Trigger2
  DriveConfiguration/Channel[1]/RealAxis/Simulation:
    SimulationModeOnPLC = SetValueGeneration
    SimulationModeOnACOPOS = NotUsed
  DriveConfiguration/Channel[2]/RealAxis:
    AxisReference = gAxisQ2
  DriveConfiguration/Channel[2]/RealAxis/MechanicalElements/Gearbox:
    InputIsReadOnly = 0
    Input = 1
    OutputIsReadOnly = 0
    Output = 1
  DriveConfiguration/Channel[2]/RealAxis/MechanicalElements/RotaryToLinearTransformation:
    ReferenceDistanceIsReadOnly = 0
    ReferenceDistance = 1
  DriveConfiguration/Channel[2]/RealAxis/Controller:
    ModeIsReadOnly = 0
    Mode = PositionController
  DriveConfiguration/Channel[2]/RealAxis/Controller/Mode/Position:
    ProportionalGain = 50.0
    IntegrationTime = 0.0
    PredictionTime = 0.0004
    TotalDelayTime = 0.0004
  DriveConfiguration/Channel[2]/RealAxis/Controller/Mode/Speed:
    ProportionalGainIsReadOnly = 0
    ProportionalGain = 2.0
    IntegrationTimeIsReadOnly = 0
    IntegrationTime = 0.0
    FilterTimeIsReadOnly = 0
    FilterTime = 0.0
  DriveConfiguration/Channel[2]/RealAxis/Controller/Mode/LoopFilters:
    LoopFilter1 = NotUsed
    LoopFilter2 = NotUsed
    LoopFilter3 = NotUsed
  DriveConfiguration/Channel[2]/RealAxis/Homing:
    Mode = Direct
  DriveConfiguration/Channel[2]/RealAxis/Homing/Mode:
    Position = 0.0
    ReferencePulse = NotUsed
  DriveConfiguration/Channel[2]/RealAxis/Homing:
    RestorePositionVariable = 
  DriveConfiguration/Channel[2]/RealAxis/StopReaction:
    Quickstop = DecelerationLimit
    DriveError = DecelerationLimit
  DriveConfiguration/Channel[2]/RealAxis/MovementErrorLimits:
    PositionError = 1.0
    VelocityErrorMonitoring = Automatic1
  DriveConfiguration/Channel[2]/RealAxis:
    JerkFilter = NotUsed
  DriveConfiguration/Channel[2]/RealAxis/DigitalInputs/HomingSwitch:
    Source = NotUsed
    Level = High
  DriveConfiguration/Channel[2]/RealAxis/DigitalInputs/PositiveLimitSwitch:
    Source = NotUsed
    Level = High
  DriveConfiguration/Channel[2]/RealAxis/DigitalInputs/NegativeLimitSwitch:
    Source = NotUsed
    Level = High
  DriveConfiguration/Channel[2]/RealAxis/DigitalInputs/Trigger1:
    Source = X8Trigger1
    Level = High
  DriveConfiguration/Channel[2]/RealAxis/DigitalInputs/Trigger2:
    Source = X8Trigger2
    Level = High
  DriveConfiguration/Channel[2]/RealAxis/DigitalInputs/Quickstop:
    Input = Trigger2
  DriveConfiguration/Channel[2]/RealAxis/Simulation:
    SimulationModeOnPLC = SetValueGeneration
    SimulationModeOnACOPOS = NotUsed
  DriveConfiguration/Channel[3]/RealAxis:
    AxisReference = gAxisQ3
  DriveConfiguration/Channel[3]/RealAxis/MechanicalElements/Gearbox:
    InputIsReadOnly = 0
    Input = 1
    OutputIsReadOnly = 0
    Output = 1
  DriveConfiguration/Channel[3]/RealAxis/MechanicalElements/RotaryToLinearTransformation:
    ReferenceDistanceIsReadOnly = 0
    ReferenceDistance = 1
  DriveConfiguration/Channel[3]/RealAxis/Controller:
    ModeIsReadOnly = 0
    Mode = PositionController
  DriveConfiguration/Channel[3]/RealAxis/Controller/Mode/Position:
    ProportionalGain = 50.0
    IntegrationTime = 0.0
    PredictionTime = 0.0004
    TotalDelayTime = 0.0004
  DriveConfiguration/Channel[3]/RealAxis/Controller/Mode/Speed:
    ProportionalGainIsReadOnly = 0
    ProportionalGain = 2.0
    IntegrationTimeIsReadOnly = 0
    IntegrationTime = 0.0
    FilterTimeIsReadOnly = 0
    FilterTime = 0.0
  DriveConfiguration/Channel[3]/RealAxis/Controller/Mode/LoopFilters:
    LoopFilter1 = NotUsed
    LoopFilter2 = NotUsed
    LoopFilter3 = NotUsed
  DriveConfiguration/Channel[3]/RealAxis/Homing:
    Mode = Direct
  DriveConfiguration/Channel[3]/RealAxis/Homing/Mode:
    Position = 0.0
    ReferencePulse = NotUsed
  DriveConfiguration/Channel[3]/RealAxis/Homing:
    RestorePositionVariable = 
  DriveConfiguration/Channel[3]/RealAxis/StopReaction:
    Quickstop = DecelerationLimit
    DriveError = DecelerationLimit
  DriveConfiguration/Channel[3]/RealAxis/MovementErrorLimits:
    PositionError = 1.0
    VelocityErrorMonitoring = Automatic1
  DriveConfiguration/Channel[3]/RealAxis:
    JerkFilter = NotUsed
  DriveConfiguration/Channel[3]/RealAxis/DigitalInputs/HomingSwitch:
    Source = NotUsed
    Level = High
  DriveConfiguration/Channel[3]/RealAxis/DigitalInputs/PositiveLimitSwitch:
    Source = NotUsed
    Level = High
  DriveConfiguration/Channel[3]/RealAxis/DigitalInputs/NegativeLimitSwitch:
    Source = NotUsed
    Level = High
  DriveConfiguration/Channel[3]/RealAxis/DigitalInputs/Trigger1:
    Source = X8Trigger1
    Level = High
  DriveConfiguration/Channel[3]/RealAxis/DigitalInputs/Trigger2:
    Source = X8Trigger2
    Level = High
  DriveConfiguration/Channel[3]/RealAxis/DigitalInputs/Quickstop:
    Input = Trigger2
  DriveConfiguration/Channel[3]/RealAxis/Simulation:
    SimulationModeOnPLC = SetValueGeneration
    SimulationModeOnACOPOS = NotUsed
```

### Config_1.axesgroup - 5APC3100_KBU3_000/mappMotion/Robot/3AxesDeltaA/Config_1.axesgroup
```
Element g3AxDeltaA (Type=axesgroup)
  Type = PathGenAxesGroup
    ProcessingTaskClass = 1
    License = 1
    PhysicalAxes:
      JointAxes:
        JointAxis[1]:
          Name = Q1
          AxisRef = gAxisQ1
        JointAxis[2]:
          Name = Q2
          AxisRef = gAxisQ2
        JointAxis[3]:
          Name = Q3
          AxisRef = gAxisQ3
    MechanicalSystem:
      MechSysRef = MechSys_3AxDeltaA
    BasicSettings:
      ModalDataBehaviour = ResetToDefault
      GeometryPlanning:
        RoundingMode = Standard
        MaxCornerDeviation = 0.0
        MaxTangentialTransitionDeviation = 0.0
        MaxRadiusDeviation = 0.001
        WorkingPlane = XY
      TrajectoryPlanning = Basic
        LimitCheckResolution = UserDefinedTime
          Time = 0.01
        BufferTime = UserDefinedTime
          Time = 0.1
    AxesGroupFeatures:
      FeatureRef[1] = Feature_Programs
      FeatureRef[2] = Feature_Jogging
      FeatureRef[3] = Feature_Frames
  Alarms = None
```

### Config_4.axesgroupfeature - 5APC3100_KBU3_000/mappMotion/Robot/3AxesDeltaA/Config_4.axesgroupfeature
```
Element Feature_Programs (Type=axesgroupfeature)
  Type = Program
    ModalDataBehaviour = UseAxesGroupSettings
    InitialSettings:
      InterpolationTypes = LinearRapid
      PositionCoordinates = Absolute
      CircleCoordinates = Relative
      JACS_ACSProgramming = JACS
      ContourConnection = Inactive
      ProgrammingUnits = UseAxesGroupSettings
      Feedrates:
        FeedCharacteristic = StandardCharacteristic
        FeedType = Feedrate
        FeedReduction = Inactive
        FeedrateValue = 0.0
        InverseFeedrateValue = 0.0
        FeedratePerRevValue = 0.0
    DefaultLanguage = BRGCode
    Location = Default
      FileDevice = CNC_PrgDir
Element Feature_Jogging (Type=axesgroupfeature)
  Type = Jogging
Element Feature_Frames (Type=axesgroupfeature)
  Type = FrameHierarchy
    ModalDataBehaviour = UseAxesGroupSettings
    FrameHierarchy = Custom
      FramePropertyMapping:
        BCS = RobotBase
        PCS = RobotBase
        SCS1 = 
        SCS2
        SCS3
        SCS4
        SCS5
      MCS:
        Frame[1]:
          Name = RobotBase
          Type = StandardFrame
            Translation:
              X = 0.0
              Y = 0.0
              Z = 1600
            Orientation:
              Angle1 = 0.0
              Angle2 = 0.0
              Angle3 = 0.0
        Frame[2]:
          Name = TrakSync
          Type = StandardFrame
            Translation:
              X = 330
              Y = 0.0
              Z = 292.5
            Orientation:
              Angle1 = 0.0
              Angle2 = 0.0
              Angle3 = 180.0
```

### CfgAssbly.assembly - 5APC3100_KBU3_000/mappMotion/Trak/CfgAssbly.assembly
```
Element gAssembly_1 (Type=assembly)
  Tracks:
    TrackSeparation = 0.030
    Track[1]:
      Segments:
        SegmentRef[1] = ::gSeg_1
        SegmentRef[2] = ::gSeg_2
        SegmentRef[3] = ::gSeg_3
        SegmentRef[4] = ::gSeg_4
        SegmentRef[5] = ::gSeg_5
        SegmentRef[6] = ::gSeg_6
        SegmentRef[7] = ::gSeg_7
        SegmentRef[8] = ::gSeg_8
        SegmentRef[9] = ::gSeg_9
        SegmentRef[10] = ::gSeg_10
        SegmentRef[11] = ::gSeg_11
        SegmentRef[12] = ::gSeg_12
        SegmentRef[13] = ::gSeg_13
        SegmentRef[14] = ::gSeg_14
      Position = Absolute
        SegmentRef = ::gSeg_1
        SegmentCountDirection = RightToLeft
        Translation:
          X = 0.0
          Y = 0.0
          Z = 0.0
        Orientation:
          Angle1 = 0.0
          Angle2 = 0.0
          Angle3 = 0.0
  CommonSegmentSettings:
    SegmentSimulationOnPLC = Off
    StopReaction = InductionHalt
    SpeedFilter = NotUsed
    ControllerParameters:
      DefaultParameter:
        Controller:
          Position:
            ProportionalGain = 0.0
          Speed:
            ProportionalGain = 0.0
            IntegrationTime = 0.0
          FeedForward:
            TotalMass = 0.0
            ForcePositive = 0.0
            ForceNegative = 0.0
            SpeedForceFactor = 0.0
            ForceLoad = 0.0
        MovementErrorLimits:
          PositionError = 0.0
          VelocityError = 0.0
      AdditionalParameterSets = NotUsed
  Shuttles:
    MaxShuttleCount = 10
    DistanceReserve:
      Collision = 0.002
      ErrorStop = 0.006
    ShuttleStereotypes:
      ShuttleStRef[1] = ShuttleStereotype_1
    MagnetPlateConfigurations:
      ShuttleType[1] = 8F1SA.100.xxxxxx-x
    CollisionAvoidance:
      Strategy = Constant
      MaximumModelDimensions:
        Length:
          ExtentToFront = 0.025
          ExtentToBack = 0.025
        Width:
          Width = 0.046
  Visualization:
    MonitoringPv = ::gShuttleMon
    ProcessingTaskClass = 1
```

### CfgProcPt.processpointlist - 5APC3100_KBU3_000/mappMotion/Trak/CfgProcPt.processpointlist
```
Element ProcessPointList_1 (Type=processpointlist)
  ProcessPoint[0]:
    Name = ppSyncStart
    SectorRef = secSync
    Position = 0.15
    TriggerEventBufferSize = 10
    BarrierFunctionality = Off
  ProcessPoint[1]:
    Name = ppSyncEnd
    SectorRef = secSync
    Position = 0.15
    PositionRelativeTo = FromEnd
    TriggerEventBufferSize = 10
    BarrierFunctionality = Off
```

### CfgSector.sector - 5APC3100_KBU3_000/mappMotion/Trak/CfgSector.sector
```
Element secStartup (Type=sector)
  Type = Composed
    StartSegment:
      SegmentRef = ::gSeg_7
    EndSegment:
      SegmentRef = ::gSeg_8
      PositionRelativeTo = FromEnd
Element secSync (Type=sector)
  Type = Composed
    StartSegment:
      SegmentRef = ::gSeg_14
      Position = 0.33
    EndSegment:
      SegmentRef = ::gSeg_1
      Position = 0.33
```

### CfgShuttle.shuttlestereotype - 5APC3100_KBU3_000/mappMotion/Trak/CfgShuttle.shuttlestereotype
```
Element ShuttleStereotype_1 (Type=shuttlestereotype)
  MeasurementUnit = 5067858
  MeasurementResolution = 0.00001
  MovementLimits = Internal
    VelocityIsReadOnly = 0
    Velocity:
      Velocity = 4.0
    AccelerationIsReadOnly = 0
    Acceleration:
      Acceleration = 50.0
    DecelerationIsReadOnly = 0
    Deceleration:
      Deceleration = 50.0
  JerkFilter = Used
    JerkTime = 0.02
  UserData:
    Size = 36
```

- Safety project (password-protected, skipped)

## Logical view

Binary libraries used (declarations not repeated): operator, runtime, astime, AsIecCon, standard, McAcp6D, AsMath, AsXml, MTBasics 5.13.0, AsBrStr, AsIODiag, LoggingLib 2.30.1, asstring, ArEventLog, AsTCP, FileIO, snprintf 1.10.2, brsystem, AsZip, MTTypes 1.03.4, sys_lib, CoTrace, MpBase, McBase 5.13.2, McAcpAx 5.13.2, McPathGen 5.13.2, McAcpTrak 5.13.2, McAxGroup 5.13.2, McAxis 5.13.2, McProgInt 5.13.2, MpRobotics 5.13.2, MpAudit

### README.md
```markdown
# Application Overview

Shuttles need to move between the following Stations
1. Load
2. Powder
3. Print
4. Tamp
5. Offload

Shuttles can likely repeat steps 2-3 numerous times before requiring to go on to the tamp process.
There are two powder depositions areas available and the shuttle can go to either

Startup positions will just be auto-driven to
    How do i start the process from the auto-drive positions?

## Robot Demo
Demo has shuttles integrate with a Delta robot to preform a "picking" or "placing" synchronization

Steps:
1. Shuttles move to recovery position (general position)
2. Send shuttle to load position, when there, sync to virtual master
3. Robot preforms movement to virtual master, shuttle is also tied. becomes synchronized
4. Shuttle then just moves in a circle back to the start to repeat

## Weighing Demo
Demo has just a basic mechanism to showcase the weighing functionality on a shuttle

1. move shuttle to defined location, wait for commands to "land" or "levitate" shuttles
2. Displays weight on HMI

# Architecture
## Shuttles
Shuttles are given a standard state machine
- Off
- Init
- Idle
- Startup
- MoveToLoad
- Load
- Error

Cmd
  - Recover
  - NextStep
Pars

Config
- LoadToPrintMacroID
- DoseToPrintMacroID
- PrintToDose1MacroID
- PrintToDose2MacroID
- DoseToPrintMacroID
- PrintToTampMacroID
- TampToUnloadMacroID
- UnloadToLoadMacroID

Status
- CurrentStep
- Destination

## Stations
Stations will wait to receive a shuttle present command/flag from a shuttle before beginning their operation

- Cmd
  - Enable
  - Process
  - Reset
- Par
  - ShuttleID
  - WaitTime
  - (Station Specific Parameters)
    - IndexRate
    - IndexAmount
    - SpinAmount
    - etc..
- Config
  - StationPos
    - X
    - Y
- Status
  - Processing
  - Done
  - Waiting
```

### Segments.var - Global variables
```iecst
VAR
	gSeg_1 : McSegmentType;
	gSeg_2 : McSegmentType;
	gSeg_3 : McSegmentType;
	gSeg_4 : McSegmentType;
	gSeg_5 : McSegmentType;
	gSeg_6 : McSegmentType;
	gSeg_7 : McSegmentType;
	gSeg_8 : McSegmentType;
	gSeg_9 : McSegmentType;
	gSeg_10 : McSegmentType;
	gSeg_11 : McSegmentType;
	gSeg_12 : McSegmentType;
	gSeg_13 : McSegmentType;
	gSeg_14 : McSegmentType;
END_VAR
```

### Package Logical/Libraries - Global libraries

### Library Logical/Libraries/WFilter (ANSIC, version 0.09.0)
Depends on: astime

#### Types.typ - Exported data types
```iecst
TYPE
	WFLowPassInternalType : 	STRUCT  (*Internal state of low pass filter*)
		input : REAL; (*Filter input*)
		level : REAL; (*Filter level*)
		state : REAL; (*Filter state*)
		output : REAL; (*Filter output*)
	END_STRUCT;
	WFMovAvgInternalType : 	STRUCT  (*Internal state of moving average filter*)
		input : REAL; (*Filter input*)
		samples : UDINT; (*Number of samples to average over*)
		state : WFMovAvgInternalBufferType; (*Internal state of moving average filter buffer*)
		error : INT; (*Equal to 1 if the buffer size is too small*)
		output : REAL; (*Filter output*)
	END_STRUCT;
	WFMovAvgInternalBufferType : 	STRUCT  (*Internal state of moving average filter buffer*)
		state : WFMovAvgInternalBufferStateType; (*Internal state of moving average filter buffer state*)
		output : REAL; (*Buffer output*)
	END_STRUCT;
	WFMovAvgInternalBufferStateType : 	STRUCT  (*Internal state of moving average filter buffer state*)
		read : UDINT; (*The buffer read position*)
		write : UDINT; (*The buffer write position*)
	END_STRUCT;
	WFPredictIntType : 	STRUCT  (*Internal state of the predictive filter*)
		input : REAL; (*Filter input*)
		t : REAL; (*Filter time constant*)
		sigma_a : REAL; (*Filter Sigma A value*)
		sigma_z : REAL; (*Filter Sigma Z value*)
		alpha : REAL; (*Filter alpha value*)
		internal : WFPredictIntInternalType; (*Internal state within the internal state of the predictive filter*)
		state : WFPredictIntStateType; (*State of the internal state within the predictive filter*)
		output : REAL; (*Filter output*)
		velocity : REAL; (*Filter velocity output*)
	END_STRUCT;
	WFPredictIntInternalType : 	STRUCT  (*Internal state within the internal state of the predictive filter*)
		t : REAL; (*Filter time constant*)
		sigma_a : REAL; (*Filter Sigma A value*)
		sigma_z : REAL; (*Filter Sigma Z value*)
		alpha : REAL; (*Filter alpha value*)
		Q : ARRAY[0..1,0..1]OF REAL; (*Filter observation noise covariance Q*)
		RR : REAL; (*Filter process noise covariance R*)
		F : ARRAY[0..1,0..1]OF REAL; (*Filter state transition model F*)
	END_STRUCT;
	WFPredictIntStateType : 	STRUCT  (*State of the internal state within the predictive filter*)
		x : ARRAY[0..1]OF REAL; (*Posterior state estimate vector x*)
		P : ARRAY[0..1,0..1]OF REAL; (*Posterior covariance matrix P*)
	END_STRUCT;
	WFFitParType : 	STRUCT  (*Parameters for fit function blocks*)
		MaxIterations : UINT; (*The maximum number of iterations to run through per cycle*)
		MaxTime : TIME; (*The maximum amount of time to run per cycle*)
	END_STRUCT;
	WFFitInternalType : 	STRUCT  (*Internal state of the fit function block*)
		x : REAL; (*X value*)
		y : REAL; (*Y value*)
		state : WFFitInternalStateType; (*State of the internal state of the fit function block*)
		a : REAL; (*A value*)
		b : REAL; (*B value*)
	END_STRUCT;
	WFFitInternalStateType : 	STRUCT  (*State of the internal state of the fit function block*)
		sumx : REAL; (*Running sum of the x values*)
		sumx2 : REAL; (*Running sum of x^2*)
		sumy : REAL; (*Running sum of the y values*)
		sumxy : REAL; (*Running sum of x*y*)
		n : UDINT; (*Number of values*)
	END_STRUCT;
	WFFitStateEnum :
		( (*State of the fit calculation*)
		wfFIT_STATE_WAIT, (*Wait to start calculation*)
		wfFIT_STATE_PROCESS (*Perform calculation*)
		);
END_TYPE
```

#### Constants.var - Exported constants
```iecst
VAR CONSTANT
	wfERR_NONE : UINT := 0; (*No error on the function block*)
	wfERR_NULLPOINTER : UINT := 1; (*The buffer points to Null*)
	wfERR_BUFFER_OVERFLOW : UINT := 2; (*The buffer is too small*)
	wfERR_ZERO_LENGTH : UINT := 3; (*The sample size is zero*)
	wfERR_FIT_CALCULATION : UINT := 4; (*Fit could not be calculated*)
END_VAR
```

#### WFilter.fun - Exported functions and function blocks
```iecst
FUNCTION_BLOCK WFLowPass (*Low Pass Filter*)
	VAR_INPUT
		Enable : BOOL; (*Enable the function block*) (* *) (*#PAR*)
		Input : REAL; (*Filter input value*) (* *) (*#CYC*)
		Level : REAL; (*Filter level*) (* *) (*#PAR*)
	END_VAR
	VAR_OUTPUT
		Active : BOOL; (*The function block is active*) (* *) (*#PAR*)
		Output : REAL; (*Filter output value*) (* *) (*#CYC*)
	END_VAR
	VAR
		Internal : WFLowPassInternalType; (*Internal state*)
		iEnable : BOOL; (*Previously recorded enable level*)
	END_VAR
END_FUNCTION_BLOCK

FUNCTION_BLOCK WFMovingAverage (*Moving Average Filter*)
	VAR_INPUT
		Enable : BOOL; (*Enable the function block*) (* *) (*#PAR*)
		Input : REAL; (*Filter input value*) (* *) (*#CYC*)
		Samples : UDINT; (*Number of samples to average over*) (* *) (*#PAR*)
		pBuffer : UDINT; (*Pointer to the sample buffer*) (* *) (*#PAR*)
		BufferSize : UDINT; (*Size of the sample buffer*) (* *) (*#PAR*)
	END_VAR
	VAR_OUTPUT
		Active : BOOL; (*The function block is active*) (* *) (*#PAR*)
		Error : BOOL; (*The function block has an error*) (* *) (*#PAR*)
		ErrorID : UINT; (*Function block error ID*) (* *) (*#PAR*)
		Output : REAL; (*Filter output value*) (* *) (*#CYC*)
		RequiredBufferSize : UDINT; (*Required size of the sample buffer*) (* *) (*#CMD*)
	END_VAR
	VAR
		Internal : WFMovAvgInternalType; (*Internal state*)
		ipBuffer : UDINT; (*Sample buffer pointer on enable*)
		iBufferSize : UDINT; (*Sample buffer size on enable*)
		iEnable : BOOL; (*Previously recorded enable level*)
	END_VAR
END_FUNCTION_BLOCK

FUNCTION_BLOCK WFPredictiveFilter (*Predictive Filter*)
	VAR_INPUT
		Enable : BOOL; (*Enable the function block*) (* *) (*#PAR*)
		Input : REAL; (*Filter input value*) (* *) (*#CYC*)
		Time : REAL; (*Time cyclic value*) (* *) (*#PAR*)
		SigmaA : REAL; (*Sigma A value*) (* *) (*#PAR*)
		SigmaZ : REAL; (*Sigma Z value*) (* *) (*#PAR*)
		Alpha : REAL; (*Fading memory alpha value*)
	END_VAR
	VAR_OUTPUT
		Active : BOOL; (*The function block is active*) (* *) (*#PAR*)
		Output : REAL; (*Filter output value*) (* *) (*#CYC*)
		ChangeRate : REAL; (*Filter output rate of change*) (* *) (*#CYC*)
	END_VAR
	VAR
		Internal : WFPredictIntType; (*Internal state*)
		iEnable : BOOL; (*Previously recorded enable level*)
	END_VAR
END_FUNCTION_BLOCK

FUNCTION_BLOCK WFLinearFit (*Linear fit of y = ax + b*)
	VAR_INPUT
		Execute : BOOL; (*Execute on rising edge*) (* *) (*#PAR*)
		Par : WFFitParType; (*Parameters for calculating the fit*) (* *) (*#PAR*)
		pDataX : UDINT; (*Pointer to the array of floats*) (* *) (*#PAR*)
		pDataY : UDINT; (*Pointer to the array of floats*) (* *) (*#PAR*)
		DataSize : UDINT; (*Size of the array of floats*) (* *) (*#PAR*)
	END_VAR
	VAR_OUTPUT
		Done : BOOL; (*Calculation of fit is complete*) (* *) (*#PAR*)
		Busy : BOOL; (*The function block is busy and needs to be continued to be called*) (* *) (*#PAR*)
		Error : BOOL; (*The function block has an error*) (* *) (*#PAR*)
		ErrorID : UINT; (*Function block error ID*) (* *) (*#PAR*)
		A : REAL; (*The A value*) (* *) (*#PAR*)
		B : REAL; (*The B value*) (* *) (*#PAR*)
	END_VAR
	VAR
		State : WFFitStateEnum; (*State of the fit calculation*)
		Counter : UDINT; (*Current position in processing data arrays*)
		Internal : WFFitInternalType; (*Internal state of the fit*)
		ipDataX : UDINT; (*DataX pointer on execute*)
		ipDataY : UDINT; (*DataY pointer on execute*)
		iDataSize : UDINT; (*Data size on execute*)
		iExecute : BOOL; (*Previously recorded execute level*)
	END_VAR
END_FUNCTION_BLOCK

FUNCTION_BLOCK WFExponentialFit (*Exponential fit of y = a*e^bx*)
	VAR_INPUT
		Execute : BOOL; (*Execute on rising edge*) (* *) (*#PAR*)
		Par : WFFitParType; (*Parameters for calculating the fit*) (* *) (*#PAR*)
		pDataX : UDINT; (*Pointer to the array of floats*) (* *) (*#PAR*)
		pDataY : UDINT; (*Pointer to the array of floats*) (* *) (*#PAR*)
		DataSize : UDINT; (*Size of the array of floats*) (* *) (*#PAR*)
	END_VAR
	VAR_OUTPUT
		Done : BOOL; (*Calculation of fit is complete*) (* *) (*#PAR*)
		Busy : BOOL; (*The function block is busy and needs to be continued to be called*) (* *) (*#PAR*)
		Error : BOOL; (*The function block has an error*) (* *) (*#PAR*)
		ErrorID : UINT; (*Function block error ID*) (* *) (*#PAR*)
		A : REAL; (*The A value*) (* *) (*#PAR*)
		B : REAL; (*The B value*) (* *) (*#PAR*)
	END_VAR
	VAR
		State : WFFitStateEnum; (*State of the fit calculation*)
		Counter : UDINT; (*Current position in processing data arrays*)
		Internal : WFFitInternalType; (*Internal state of the fit*)
		ipDataX : UDINT; (*DataX pointer on execute*)
		ipDataY : UDINT; (*DataY pointer on execute*)
		iDataSize : UDINT; (*Data size on execute*)
		iExecute : BOOL; (*Previously recorded execute level*)
	END_VAR
END_FUNCTION_BLOCK
```

#### filter_fub.c - Filter function blocks
```c
#include <bur/plctypes.h>
#include <astime.h>
#include <WFilter.h>
#include "filter.h"

void WFLowPass(struct WFLowPass* inst){

    lowpass_typ* internalptr = (lowpass_typ*) &inst->Internal;

    // Update the level and reset the state
    // on a positive edge of the enable
    if(inst->Enable & !inst->iEnable){
        inst->Internal.level = inst->Level;
        inst->Internal.state = 0.0;
    }
    inst->iEnable = inst->Enable;
    inst->Active = inst->Enable;

    // Update the values only while enable is true,
    // otherwise return 0
    if(inst->Enable){
        inst->Internal.input = inst->Input;
        lowpass(internalptr);
        inst->Output = inst->Internal.output;
    }
    else{
        inst->Output = 0.0;
    }

}

void WFMovingAverage(struct WFMovingAverage* inst){

    float* bufferptr;
    mov_avg_typ* internalptr = (mov_avg_typ*) &inst->Internal;

    // Update the data and reset the state
    // on a positive edge of the enable
    if(inst->Enable & !inst->iEnable){
        memset(&inst->Internal, 0, sizeof(inst->Internal));
        inst->Internal.samples = inst->Samples;
        inst->ipBuffer = inst->pBuffer;
        inst->iBufferSize = inst->BufferSize;
    }
    inst->iEnable = inst->Enable;

    // Update the values only while enable is true,
    // otherwise return 0
    if(inst->Enable){
        if(inst->ipBuffer){
            if(inst->Internal.samples){
                bufferptr = (float*) inst->ipBuffer;
                inst->Internal.input = inst->Input;
                mov_avg(internalptr, bufferptr, inst->iBufferSize);
                if(inst->Internal.error){
                    inst->Output = 0.0;
                    inst->ErrorID = wfERR_BUFFER_OVERFLOW;
                    inst->Active = 1;
                }
                else{
                    inst->Output = inst->Internal.output;
                    inst->Error = 0;
                    inst->ErrorID = wfERR_NONE;
                    inst->Active = 0;
                }
            }
            else{
                inst->Output = 0.0;
                inst->Error = 1;
                inst->ErrorID = wfERR_ZERO_LENGTH;
                inst->Active = 0;
            }
        }
        else{
            inst->Output = 0.0;
            inst->Error = 1;
            inst->ErrorID = wfERR_NULLPOINTER;
            inst->Active = 0;
        }
        inst->RequiredBufferSize = (inst->Internal.samples + 2) * sizeof(float);
    }
    else{
        inst->Output = 0.0;
        inst->Error = 0;
        inst->ErrorID = wfERR_NONE;
        inst->Active = 0;
        inst->RequiredBufferSize = 0;
    }

}

void WFPredictiveFilter(struct WFPredictiveFilter* inst){

    kalman_typ* internalptr = (kalman_typ*) &inst->Internal;

    // Update the data and reset the state
    // on a positive edge of the enable
    if(inst->Enable & !inst->iEnable){
        memset(&inst->Internal, 0, sizeof(inst->Internal));
        inst->Internal.t = inst->Time;
        inst->Internal.sigma_a = inst->SigmaA;
        inst->Internal.sigma_z = inst->SigmaZ;
		inst->Internal.alpha = inst->Alpha;
        inst->Internal.state.x[0] = inst->Input;
    }
    inst->iEnable = inst->Enable;
    inst->Active = inst->Enable;

    // Update the values only while enable is true,
    // otherwise return 0
    if(inst->Enable){
        inst->Internal.input = inst->Input;
        kalman(internalptr);
        inst->Output = inst->Internal.output;
        inst->ChangeRate = inst->Internal.velocity;
    }
    else{
        inst->Output = 0.0;
        inst->ChangeRate = 0.0;
    }

}

void WFLinearFit(struct WFLinearFit* inst){

    fit_typ* internalptr = (fit_typ*) &inst->Internal;
    float* dataptr;

    short continue_process;
    unsigned long iteration_number;
    signed long start_time;
    signed long current_time;
    signed long elapsed_time;
    int status;

    signed long total_length = inst->DataSize / sizeof(float);

    switch(inst->State){

        case wfFIT_STATE_WAIT:

            //The function block is not busy
            inst->Busy = 0;

            //Reset the Done bit and errors when the execute signal goes low
            if(!inst->Execute){
                inst->Done = 0;
                inst->Error = 0;
                inst->ErrorID = wfERR_NONE;
            }

            //Check for execute command and copy parameters
            if(inst->Execute & !inst->iExecute){
                //The function block is busy
                inst->Busy = 1;
                inst->ipDataX = inst->pDataX;
                inst->ipDataY = inst->pDataY;
                inst->iDataSize = inst->DataSize;
                inst->Counter = 0;
                linearfitinit(internalptr);
                if(inst->ipDataX & inst->ipDataY){
                    if(inst->iDataSize){
                        inst->State = wfFIT_STATE_PROCESS;
                    }
                    else{
                        inst->Error = 1;
                        inst->ErrorID = wfERR_ZERO_LENGTH;
                    }
                }
                else{
                    inst->Error = 1;
                    inst->ErrorID = wfERR_NULLPOINTER;
                }
            }

            break;

        case wfFIT_STATE_PROCESS:

            //Reset the iteration number and start time
            iteration_number = 0;
            start_time = clock_ms();
            elapsed_time = 0;

            do{

                //Get the data values
                dataptr = (float*) inst->ipDataX;
                inst->Internal.x = dataptr[inst->Counter];
                dataptr = (float*) inst->ipDataY;
                inst->Internal.y = dataptr[inst->Counter];
                status = linearfitupdate(internalptr);

                if(status){
                    inst->Error = 1;
                    inst->ErrorID = wfERR_FIT_CALCULATION;
                    inst->State = wfFIT_STATE_WAIT;
                }

                //Increment the counter, iteration number, and time
                inst->Counter += 1;
                iteration_number += 1;
                current_time = clock_ms();
                elapsed_time = current_time - start_time;

                //Check for completion
                if(inst->Counter >= total_length){
                    status = linearfitfinal(internalptr);
                    if(status){
                        inst->Error = 1;
                        inst->ErrorID = wfERR_FIT_CALCULATION;
                    }
                    if(!inst->Error){
                        //Return results if error-free
                        inst->A = inst->Internal.a;
                        inst->B = inst->Internal.b;
                        inst->Done = 1;
                    }
                    inst->State = wfFIT_STATE_WAIT;
                }

                continue_process = (iteration_number < inst->Par.MaxIterations) &
                                   (elapsed_time < inst->Par.MaxTime) &
                                   (inst->Counter < total_length) &
                                   !inst->Error;

            }while(continue_process);

            break;

    }

    inst->iExecute = inst->Execute;

}

void WFExponentialFit(struct WFExponentialFit* inst){

    fit_typ* internalptr = (fit_typ*) &inst->Internal;
    float* dataptr;

    short continue_process;
    unsigned long iteration_number;
    signed long start_time;
    signed long current_time;
    signed long elapsed_time;
    int status;

    signed long total_length = inst->DataSize / sizeof(float);

    switch(inst->State){

        case wfFIT_STATE_WAIT:

            //The function block is not busy
            inst->Busy = 0;

            //Reset the Done bit and errors when the execute signal goes low
            if(!inst->Execute){
                inst->Done = 0;
                inst->Error = 0;
                inst->ErrorID = wfERR_NONE;
            }

            //Check for execute command and copy parameters
            if(inst->Execute & !inst->iExecute){
                //The function block is busy
                inst->Busy = 1;
                inst->ipDataX = inst->pDataX;
                inst->ipDataY = inst->pDataY;
                inst->iDataSize = inst->DataSize;
                inst->Counter = 0;
                exponentialfitinit(internalptr);
                if(inst->ipDataX & inst->ipDataY){
                    if(inst->iDataSize){
                        inst->State = wfFIT_STATE_PROCESS;
                    }
                    else{
                        inst->Error = 1;
                        inst->ErrorID = wfERR_ZERO_LENGTH;
                    }
                }
                else{
                    inst->Error = 1;
                    inst->ErrorID = wfERR_NULLPOINTER;
                }
            }

            break;

        case wfFIT_STATE_PROCESS:

            //Reset the iteration number and start time
            iteration_number = 0;
            start_time = clock_ms();
            elapsed_time = 0;

            do{

                //Get the data values
                dataptr = (float*) inst->ipDataX;
                inst->Internal.x = dataptr[inst->Counter];
                dataptr = (float*) inst->ipDataY;
                inst->Internal.y = dataptr[inst->Counter];
                status = exponentialfitupdate(internalptr);

                if(status){
                    inst->Error = 1;
                    inst->ErrorID = wfERR_FIT_CALCULATION;
                    inst->State = wfFIT_STATE_WAIT;
                }

                //Increment the counter, iteration number, and time
                inst->Counter += 1;
                iteration_number += 1;
                current_time = clock_ms();
                elapsed_time = current_time - start_time;

                //Check for completion
                if(inst->Counter >= total_length){
                    status = exponentialfitfinal(internalptr);
                    if(status){
                        inst->Error = 1;
                        inst->ErrorID = wfERR_FIT_CALCULATION;
                    }
                    if(!inst->Error){
                        //Return results if error-free
                        inst->A = inst->Internal.a;
                        inst->B = inst->Internal.b;
                        inst->Done = 1;
                    }
                    inst->State = wfFIT_STATE_WAIT;
                }

                continue_process = (iteration_number < inst->Par.MaxIterations) &
                    (elapsed_time < inst->Par.MaxTime) &
                    (inst->Counter < total_length) &
                    !inst->Error;

            }while(continue_process);

            break;

    }

    inst->iExecute = inst->Execute;

}
```

#### filter.c - Filter functions
```c
/*
 ============================================================================
 Name        : filter.c
 Author      : B&R Industrial Automation
 Version     :
 Copyright   :
 Description : Filter programs
 ============================================================================
 */

#include "filter.h"

BUILD_DLL int lowpass(struct lowpass* inst) {
	/*
	 * Implements a low pass filter
	*/
    float levelfactor;
    levelfactor = (float)(1.0 / (pow(2.0, (double) inst->level)));
    inst->output = ((inst->input - inst->state) * levelfactor) + inst->state;
    inst->state = inst->output;
    return 0;
}

int buflen(bufferstate_typ* bufferstate, unsigned long maxlen) {
	/*
	 * Returns the current length of the ring buffer
	*/
    int length;
    length = bufferstate->write - bufferstate->read;
    if(length < 0) {
        length += maxlen;
    }
    return length;
}

int bufappend(bufferstate_typ* bufferstate, float* buffer, unsigned long maxlen, float value) {
	/*
	 * Append a value to the ring buffer
	*/
    buffer[bufferstate->write] = value;
    bufferstate->write = (bufferstate->write + 1) % maxlen;
    return 0;
}

float bufpop(bufferstate_typ* bufferstate, float* buffer, unsigned long maxlen) {
	/*
	 * Returns and removes the first item from the ring buffer
	*/
    float value;
    value = buffer[bufferstate->read];
    bufferstate->read = (bufferstate->read + 1) % maxlen;
    return value;
}

BUILD_DLL int mov_avg(struct mov_avg* inst, float* buffer, unsigned long bufferlen) {
	/*
	 * Implements a moving average filter
	*/
    float divval;
    unsigned long maxlen = bufferlen / sizeof(float);

    if(maxlen < (inst->samples + 2)) {
        inst->error = 1;
        return 1;
    }
    else {
        inst->error = 0;
    }

    if(inst->samples > 0) {
        divval = inst->input / inst->samples;
        bufappend(&inst->state.bufferstate, buffer, maxlen, divval);
        if (buflen(&inst->state.bufferstate, maxlen) > inst->samples) {
            divval -= bufpop(&inst->state.bufferstate, buffer, maxlen);
        }
        divval += inst->state.output;
        inst->output = divval;
        inst->state.output = divval;
    }
    return 0;
}

float second_order_fir(float input, float a[2], float b[3], second_order_fir_state_typ* state) {
	/*
	 * Implements a second order FIR filter
	*/
    float output;

    output = (input * b[0]) + (state->input[0] * b[1]) + (state->input[1] * b[2]) +
        (state->output[0] * a[0]) + (state->output[1] * a[1]);

    state->input[1] = state->input[0];
    state->input[0] = input;

    state->output[1] = state->output[0];
    state->output[0] = output;

    return output;
}

float cascade_fir(float input, float a[4][2], float b[4][3], second_order_fir_state_typ state[4]) {
	/*
	 * Implements a cascade of four second order FIR filters
	*/
int i;
float intermediate[4];

for(i = 0; i < 4; i++) {

        if(i > 0) {
intermediate[i] = second_order_fir(intermediate[i - 1], a[i], b[i], state + i);
        }
        else {
intermediate[i] = second_order_fir(input, a[i], b[i], state + i);
        }

    }

return intermediate[3];
}

BUILD_DLL int notch_fir(struct notch_fir* inst) {
	/*
	 * Implements a notch filter using a cascade of four second order FIR filters
	*/
    float a_50Hz_40dB[4][2] = {{1.993991099002, -0.997449015889},
        {1.992719432869, -0.997122121373},
        {1.989918295292, -0.993622497931},
        {1.989201706440, -0.993295984254}
        };

    float a_50Hz_60dB[4][2] = {{1.993792556381, -0.997261542221},
        {1.992532991646, -0.996920780978},
        {1.989453530594, -0.993161909468},
        {1.988733858877, -0.992821608511}
        };

    float a_50Hz_80dB[4][2] = {{1.993728075618, -0.997200655249},
        {1.992472700971, -0.996855673897},
        {1.989302815679, -0.993012548252},
        {1.988582415484, -0.992668052597}
        };

    float a_60Hz_40dB[4][2] = {{1.992325153524, -0.997421548427},
        {1.990918758069, -0.997149580589},
        {1.988199921793, -0.993594951604},
        {1.987460059960, -0.993323522293}
        };

    float a_60Hz_60dB[4][2] = {{1.992123011711, -0.997232903629},
        {1.990736250797, -0.996949410606},
        {1.987733301547, -0.993133190117},
        {1.986994878892, -0.992850318851}
        };

    float a_60Hz_80dB[4][2] = {{1.992057387679, -0.997171660034},
        {1.990677211885, -0.996884659925},
        {1.987582008256, -0.992983471531},
        {1.986844276615, -0.992697120082}
        };

    float b_50Hz_40dB[4][3] = {{0.997682591232, -1.991694270059, 0.997682591232},
        {0.997682591232, -1.991225875619, 0.997682591232},
        {0.997682591232, -1.991562861801, 0.997682591232},
        {0.997682591232, -1.991368918450, 0.997682591232}
        };

    float b_50Hz_60dB[4][3] = {{0.997516583626, -1.991267524831, 0.997516583626},
        {0.997516583626, -1.990999323659, 0.997516583626},
        {0.997516583626, -1.991190872529, 0.997516583626},
        {0.997516583626, -1.991079793498, 0.997516583626}
        };

    float b_50Hz_80dB[4][3] = {{0.997462788341, -1.991103458477, 0.997462788341},
        {0.997462788341, -1.990951762853, 0.997462788341},
        {0.997462788341, -1.991059637418, 0.997462788341},
        {0.997462788341, -1.990996805483, 0.997462788341}
        };

    float b_60Hz_40dB[4][3] = {{0.997682591234, -1.990009760159, 0.997682591234},
        {0.997682591234, -1.989447061155, 0.997682591234},
        {0.997682591234, -1.989850731814, 0.997682591234},
        {0.997682591234, -1.989617713958, 0.997682591234}
        };

    float b_60Hz_60dB[4][3] = {{0.997516583631, -1.989563160946, 0.997516583631},
        {0.997516583631, -1.989240931265, 0.997516583631},
        {0.997516583631, -1.989470683554, 0.997516583631},
        {0.997516583631, -1.989337222874, 0.997516583631}
        };

    float b_60Hz_80dB[4][3] = {{0.997462788347, -1.989387454539, 0.997462788347},
        {0.997462788347, -1.989205194537, 0.997462788347},
        {0.997462788347, -1.989334681058, 0.997462788347},
        {0.997462788347, -1.989259188525, 0.997462788347}
        };

    switch(inst->mode) {

        case 0: //50 Hz, 40 dB
            inst->output = cascade_fir(inst->input, a_50Hz_40dB, b_50Hz_40dB, inst->state);
            break;

        case 1: //50 Hz, 60 dB
            inst->output = cascade_fir(inst->input, a_50Hz_60dB, b_50Hz_60dB, inst->state);
            break;

        case 2: //50 Hz, 80 dB
            inst->output = cascade_fir(inst->input, a_50Hz_80dB, b_50Hz_80dB, inst->state);
            break;

        case 3: //60 Hz, 40 dB
            inst->output = cascade_fir(inst->input, a_60Hz_40dB, b_60Hz_40dB, inst->state);
            break;

        case 4: //60 Hz, 60 dB
            inst->output = cascade_fir(inst->input, a_60Hz_60dB, b_60Hz_60dB, inst->state);
            break;

        case 5: //60 Hz, 80 dB
            inst->output = cascade_fir(inst->input, a_60Hz_80dB, b_60Hz_80dB, inst->state);
            break;

    }
    return 0;
}

int dot_product(float a[2][2], float b[2][2], float output[2][2]) {
	/*
	 * Take the dot product of two 2x2 matrices
	 */
output[0][0] = (a[0][0] * b[0][0]) + (a[0][1] * b[1][0]);
output[0][1] = (a[0][0] * b[0][1]) + (a[0][1] * b[1][1]);
output[1][0] = (a[1][0] * b[0][0]) + (a[1][1] * b[1][0]);
output[1][1] = (a[1][0] * b[0][1]) + (a[1][1] * b[1][1]);
	return 0;
}

int transpose(float input[2][2], float output[2][2]) {
	/*
	 * Transpose the input 2x2 matrix
	 */
output[0][0] = input[0][0];
output[0][1] = input[1][0];
output[1][0] = input[0][1];
output[1][1] = input[1][1];
	return 0;
}

int add_matrix(float a[2][2], float b[2][2], float output[2][2]) {
	/*
	 * Add two 2x2 matrices together
	 */
output[0][0] = a[0][0] + b[0][0];
output[0][1] = a[0][1] + b[0][1];
output[1][0] = a[1][0] + b[1][0];
output[1][1] = a[1][1] + b[1][1];
	return 0;
}

int scale_matrix(float a, float b[2][2], float output[2][2]) {
	/*
	 * Multiply a 2x2 matrix by a scalar
	 */
output[0][0] = a * b[0][0];
output[0][1] = a * b[0][1];
output[1][0] = a * b[1][0];
output[1][1] = a * b[1][1];
	return 0;
}

int kalman_update(float input, kalman_state_typ* state, float R) {
    /*
     * Add a new measurement input to the Kalman filter.
     *
     * Parameters
     * ----------
     * input : measurement for this update.
     * state : kalman filter state
     * R : Measurement noise matrix
    */

    float y;
    float S;
    float K[2];
    float I_KH[2][2];
    float I_KHT[2][2];
    float KRKT[2][2];
    float intermediate[2][2];
    float dot3[2][2];

    // error (residual) between measurement and prediction
    y = input - state->x[0];

    // project system uncertainty into measurement space
    S = state->P[0][0] + R;

    // map system uncertainty into kalman gain
    if(S != 0) {
        K[0] = state->P[0][0] / S;
        K[1] = state->P[1][0] / S;
    }

    // predict new x with residual scaled by the kalman gain
    state->x[0] = state->x[0] + (K[0] * y);
    state->x[1] = state->x[1] + (K[1] * y);

    // P = (I-KH)P(I-KH)' + KRK'
    I_KH[0][0] = 1 - K[0];
    I_KH[0][1] = 0;
    I_KH[1][0] = -K[1];
    I_KH[1][1] = 1;

    transpose(I_KH, I_KHT);

    KRKT[0][0] = R * K[0] * K[0];
    KRKT[0][1] = R * K[0] * K[1];
    KRKT[1][0] = R * K[0] * K[1];
    KRKT[1][1] = R * K[1] * K[1];

    dot_product(state->P, I_KHT, intermediate);
    dot_product(I_KH, intermediate, dot3);
    add_matrix(dot3, KRKT, state->P);

    return 0;

}

int kalman_predict(kalman_state_typ* state, float F[2][2], float Q[2][2], float alpha) {
    /*
     * Predict next position using the Kalman filter state propagation
     * equations.
     *
     * Parameters
     * ----------
     * state : kalman filter state
     * F : State Transition matrix
     * Q : Process noise matrix
     * alpha : Fading memory setting. 1.0 gives the normal Kalman filter, and
     *         values slightly larger than 1.0 (such as 1.02) give a fading
     *         memory effect - previous measurements have less influence on the
     *         filter's estimates. This formulation of the Fading memory filter
     *         (there are many) is due to Dan Simon
    */

	float FT[2][2];
	float intermediate[2][2];
	float dot3[2][2];

	state->x[0] = (state->x[0] * F[0][0]) + (state->x[1] * F[0][1]);
	state->x[1]	= (state->x[0] * F[1][0]) + (state->x[1] * F[1][1]);

	transpose(F, FT);
	dot_product(state->P, FT, intermediate);
    dot_product(F, intermediate, dot3);
    scale_matrix(alpha * alpha, dot3, intermediate);
    add_matrix(intermediate, Q, state->P);

    return 0;

}

BUILD_DLL int kalman(struct kalman* inst) {
	/*
	 * Implement a Kalman filter
	*/

    float intermediate[2][2];

    // Update the matrices if the inputs have changed
    if((inst->t != inst->internal.t) ||
        (inst->sigma_a != inst->internal.sigma_a) ||
    (inst->sigma_z != inst->internal.sigma_z) ||
	(inst->alpha != inst->internal.alpha)) {

        intermediate[0][0] = (float)(pow((double) inst->t, 4.0) / 4.0);
        intermediate[0][1] = (float)(pow((double) inst->t, 3.0) / 2.0);
        intermediate[1][0] = (float)(pow((double) inst->t, 3.0) / 2.0);
        intermediate[1][1] = (float)(pow((double) inst->t, 2.0));

        scale_matrix(inst->sigma_a * inst->sigma_a, intermediate, inst->internal.Q);

        inst->internal.R = inst->sigma_z * inst->sigma_z;

        inst->internal.F[0][0] = 1;
        inst->internal.F[0][1] = inst->t;
        inst->internal.F[1][0] = 0;
        inst->internal.F[1][1] = 1;

        inst->internal.t = inst->t;
        inst->internal.sigma_a = inst->sigma_a;
        inst->internal.sigma_z = inst->sigma_z;
		inst->internal.alpha = inst->alpha;

    }

    kalman_predict(&inst->state, inst->internal.F, inst->internal.Q, inst->internal.alpha);
    kalman_update(inst->input, &inst->state, inst->internal.R);

    inst->output = inst->state.x[0];
    inst->velocity = inst->state.x[1];

    return 0;
}

BUILD_DLL int linearfitinit(struct fit* inst) {
    /*
     * Initialize the reference data for a linear fit
     */
    memset(inst, 0, sizeof(*inst));

    return 0;
}

BUILD_DLL int linearfitupdate(struct fit* inst) {
    /*
     * Update the reference data for a linear fit
     */
    inst->state.n += 1;
    inst->state.sumx += inst->x;
    inst->state.sumx2 += inst->x * inst->x;
    inst->state.sumy += inst->y;
    inst->state.sumxy += inst->x * inst->y;

    return 0;
}

BUILD_DLL int linearfitfinal(struct fit* inst) {
	/*
	 * Finalize the data for a linear fit
	 * in the form of y = ax + b
	 */

    if(((inst->state.n * inst->state.sumx2) - (inst->state.sumx * inst->state.sumx))){
        inst->a = ((inst->state.n * inst->state.sumxy) - (inst->state.sumx * inst->state.sumy)) /
            ((inst->state.n * inst->state.sumx2) - (inst->state.sumx * inst->state.sumx));
    }
    else{
        inst->a = 0;
        inst->b = 0;
        return 1;
    }

    if(inst->state.n){
        inst->b = (inst->state.sumy - (inst->a * inst->state.sumx)) / inst->state.n;
    }
    else{
        inst->b = 0;
        return 1;
    }

    return 0;
}

BUILD_DLL int exponentialfitinit(struct fit* inst) {
    /*
     * Initialize the reference data for an exponential fit
     */
    memset(inst, 0, sizeof(*inst));

    return 0;
}

BUILD_DLL int exponentialfitupdate(struct fit* inst) {
    /*
     * Update the reference data for an exponential fit
     */
    float Y;

    if(inst->y > 0){
        Y = log(inst->y);

        inst->state.n += 1;
        inst->state.sumx = inst->state.sumx + inst->x;
        inst->state.sumx2 = inst->state.sumx2 + (inst->x * inst->x);
        inst->state.sumy = inst->state.sumy + Y;
        inst->state.sumxy = inst->state.sumxy + (inst->x * Y);
    }
    else{
        inst->b = 0;
        inst->a = 0;
        return 1;
    }

    return 0;
}

BUILD_DLL int exponentialfitfinal(struct fit* inst) {
	/*
	 * Finalize the data for an exponential fit
	 * in the form of y = a*e^bx
	 */
    float A;

    if(((inst->state.n * inst->state.sumx2) - (inst->state.sumx * inst->state.sumx))){
        A = ((inst->state.sumx2 * inst->state.sumy) - (inst->state.sumx * inst->state.sumxy)) /
            ((inst->state.n * inst->state.sumx2) - (inst->state.sumx * inst->state.sumx));

        inst->b = ((inst->state.n * inst->state.sumxy) - (inst->state.sumx * inst->state.sumy)) /
            ((inst->state.n * inst->state.sumx2) - (inst->state.sumx * inst->state.sumx));

        inst->a = exp(A);
    }
    else{
        inst->b = 0;
        inst->a = 0;
        return 1;
    }

    return 0;
}

int main(void) {
    return 0;
}
```

#### filter.h - Filter headers
```c
 /*
 ============================================================================
 Name        : filter.h
 Author      : B&R Industrial Automation
 Version     :
 Copyright   :
 Description : Filter program headers
 ============================================================================
 */

#ifndef WEIGH_FILTER_C_H
#define WEIGH_FILTER_C_H

#include <stdio.h>
#include <string.h>
#include <asmath.h>
//#include <math.h>

#ifdef BUILD_DLL
#define BUILD_DLL __declspec(dllexport)
#else
#define BUILD_DLL
#endif

BUILD_DLL typedef struct lowpass {
    float input;
    float level;
    float state;
    float output;
} lowpass_typ;

BUILD_DLL int lowpass(struct lowpass* inst);

typedef struct bufferstate {
    unsigned long read;
    unsigned long write;
} bufferstate_typ;

int buflen(bufferstate_typ* bufferstate, unsigned long maxlen);
int bufappend(bufferstate_typ* bufferstate, float* buffer, unsigned long maxlen, float value);
float bufpop(bufferstate_typ* bufferstate, float* buffer, unsigned long maxlen);

typedef struct mov_avg_state {
    bufferstate_typ bufferstate;
    float output;
} mov_avg_state_typ;

BUILD_DLL typedef struct mov_avg {
    float input;
    unsigned long samples;
    mov_avg_state_typ state;
    short error;
    float output;
} mov_avg_typ;

BUILD_DLL int mov_avg(struct mov_avg* inst, float* buffer, unsigned long bufferlen);

typedef struct second_order_fir_state {
    float input[2];
    float output[2];
} second_order_fir_state_typ;

float second_order_fir(float input, float a[2], float b[3], second_order_fir_state_typ* state);

float cascade_fir(float input, float a[4][2], float b[4][3], second_order_fir_state_typ state[4]);

BUILD_DLL typedef struct notch_fir {
    float input;
    int mode;
    second_order_fir_state_typ state[4];
    float output;
} notch_fir_typ;

BUILD_DLL int notch_fir(struct notch_fir* inst);

typedef struct kalman_state {
	/*
	 * x : Posterior state estimate vector
	 * P : Posterior covariance matrix
	*/
    float x[2];
    float P[2][2];
} kalman_state_typ;

int dot_product(float in1[2][2], float in2[2][2], float out[2][2]);

int kalman_update(float input, kalman_state_typ* state, float R);

int kalman_predict(kalman_state_typ* state, float F[2][2], float Q[2][2], float alpha);

typedef struct kalman_internal {
	float t;
	float sigma_a;
	float sigma_z;
	float alpha;
	float Q[2][2];
	float R;
	float F[2][2];
} kalman_internal_typ;

BUILD_DLL typedef struct kalman {
	float input;
	float t;
	float sigma_a;
	float sigma_z;
	float alpha;
	kalman_internal_typ internal;
	kalman_state_typ state;
	float output;
	float velocity;
} kalman_typ;

BUILD_DLL int kalman(struct kalman* inst);

typedef struct fit_state {
    float sumx;
    float sumx2;
    float sumy;
    float sumxy;
    unsigned long n;
} fit_state_typ;

BUILD_DLL typedef struct fit {
    float x;
    float y;
    fit_state_typ state;
    float a;
    float b;
} fit_typ;

BUILD_DLL int linearfitinit(struct fit* inst);
BUILD_DLL int linearfitupdate(struct fit* inst);
BUILD_DLL int linearfitfinal(struct fit* inst);

BUILD_DLL int exponentialfitinit(struct fit* inst);
BUILD_DLL int exponentialfitupdate(struct fit* inst);
BUILD_DLL int exponentialfitfinal(struct fit* inst);

#endif
```

### Test.st - not listed in the package file held
```iecst
VAR CONSTANT
    P : McPointType := (Pos:=(X:= 660, Y:=0 , Z:=0));
END_VAR

PROGRAM _MAIN
    Feedrate(1000*60);
    WaitTime(3);

END_PROGRAM
```

### GlobalVars.var
```iecst
(*Constants*)
VAR CONSTANT
	MAX_SHUTTLE_COUNT : USINT := 8; (*Maximum count of shuttles allowed in the system*)
	MAX_SHUTTLE_COUNT_ARRAY : USINT := MAX_SHUTTLE_COUNT-1; (*Maximum count of shuttles - 1 (used for array declaration)*)
	STATION_IS_EMPTY : USINT := 255; (*Index that denotes that a station is empty and available*)
	NUM_DOSE_STATIONS : USINT := 2; (*Number of dosing stations in the system*)
	NUM_DOSE_STATIONS_ARRAY : USINT := NUM_DOSE_STATIONS-1; (*Number of dosing stations in the system - 1 (used for array declaration)*)
END_VAR
(*Global Interfaces*)
VAR
	gShuttleIf : ARRAY[0..1] OF gShuttleIfTyp; (*Interface(s) to control shuttles in the system*)
	gAcp6DCtrlIf : Acp6DCtrlType; (*Interface to control the 6D system as a whole*)
	gMainIf : MainIfTyp := (Cfg:=(ShuttleCount:=1)); (*Main interface to control the system*)
	gLoadStationIf : LoadStationIfTyp; (*Interface to control the load station*)
	g6DRecoveryIf : Acp6DRecoveryIfTyp; (*Interface to control the recover process*)
	gProcessInfoIf : ProcessInfoIfTyp; (*Interface to display process related information*)
	gSyncIf : SyncSecIfTyp;
	gRobotIf : RobotIfTyp;
	gPickPlaceIf : RobotPickPlaceTyp;
	gSceneViewerIf : SceneViewerTyp;
END_VAR
```
